SPLINE
SPL {X  -157.921, Y  +697.149, Z    +0.000, E1  +377.701, E3 -358437.505}
SPL {X  -159.579, Y  +682.959, Z    +0.000, E1  +369.793, E3 -358445.453}
SPL {X  -159.938, Y  +675.561, Z    +0.000, E1  +365.399, E3 -358447.875}
SPL {X  -159.990, Y  +669.910, Z    +0.000, E1  +361.710, E3 -358449.166}
SPL {X  -159.990, Y  +665.465, Z    +0.000, E1  +358.378, E3 -358450.084}
SPL {X  -159.990, Y  +661.791, Z    +0.000, E1  +355.213, E3 -358450.921}
SPL {X  -159.990, Y  +656.991, Z    +0.000, E1  +350.742, E3 -358452.341}
SPL {X  -159.990, Y  +648.067, Z    +0.000, E1  +342.328, E3 -358456.070}
SPL {X  -159.990, Y  +624.891, Z    +0.000, E1  +327.004, E3 -358474.558}
SPL {X  -159.990, Y  +618.109, Z    +0.000, E1  +324.631, E3 -358482.734}
SPL {X  -159.990, Y  +591.256, Z    +0.000, E1  +319.966, E3 -358526.411}
SPL {X  -159.990, Y  +586.740, Z    +0.000, E1  +319.956, E3 -358537.801}
SPL {X  -159.990, Y  +581.814, Z    +0.000, E1  +319.956, E3 -358550.241}
SPL {X  -159.990, Y  +577.274, Z    +0.000, E1  +319.964, E3 -358561.718}
SPL {X  -159.990, Y  +572.933, Z    +0.000, E1  +319.959, E3 -358572.660}
SPL {X  -159.990, Y  +568.504, Z    +0.000, E1  +319.956, E3 -358583.822}
SPL {X  -159.990, Y  +564.427, Z    +0.000, E1  +319.959, E3 -358594.108}
SPL {X  -159.990, Y  +558.823, Z    +0.000, E1  +319.916, E3 -358608.188}
SPL {X  -159.990, Y  +553.571, Z    +0.000, E1  +319.954, E3 -358621.469}
SPL {X  -159.990, Y  +549.413, Z    +0.000, E1  +319.938, E3 -358631.935}
SPL {X  -159.990, Y  +543.439, Z    +0.000, E1  +319.921, E3 -358647.023}
SPL {X  -159.990, Y  +537.213, Z    +0.000, E1  +319.937, E3 -358662.766}
SPL {X  -159.990, Y  +532.291, Z    +0.000, E1  +319.951, E3 -358675.191}
SPL {X  -159.990, Y  +527.393, Z    +0.000, E1  +319.924, E3 -358687.500}
SPL {X  -159.990, Y  +522.533, Z    +0.000, E1  +319.951, E3 -358699.797}
SPL {X  -159.990, Y  +502.378, Z    +0.000, E1  +313.079, E3 -358704.201}
SPL {X  -159.990, Y  +493.568, Z    +0.000, E1  +312.053, E3 -358715.369}
SPL {X  -159.990, Y  +489.464, Z    +0.000, E1  +313.059, E3 -358729.235}
SPL {X  -159.990, Y  +484.831, Z    +0.000, E1  +314.066, E3 -358744.769}
SPL {X  -159.990, Y  +480.580, Z    +0.000, E1  +315.242, E3 -358760.455}
SPL {X  -159.990, Y  +476.546, Z    +0.000, E1  +316.165, E3 -358774.750}
SPL {X  -159.990, Y  +472.671, Z    +0.000, E1  +317.192, E3 -358789.577}
SPL {X  -159.990, Y  +468.809, Z    +0.000, E1  +318.343, E3 -358805.506}
SPL {X  -159.990, Y  +465.057, Z    +0.000, E1  +319.375, E3 -358820.664}
SPL {X  -159.990, Y  +461.409, Z    +0.000, E1  +319.848, E3 -358832.564}
SPL {X  -159.990, Y  +456.934, Z    +0.000, E1  +319.854, E3 -358843.839}
SPL {X  -159.990, Y  +452.940, Z    +0.000, E1  +319.854, E3 -358853.884}
SPL {X  -159.990, Y  +448.856, Z    +0.000, E1  +319.859, E3 -358864.167}
SPL {X  -159.990, Y  +444.973, Z    +0.000, E1  +319.856, E3 -358873.933}
SPL {X  -159.990, Y  +439.927, Z    +0.000, E1  +319.837, E3 -358886.589}
SPL {X  -159.990, Y  +435.246, Z    +0.000, E1  +319.853, E3 -358898.398}
SPL {X  -159.990, Y  +430.690, Z    +0.000, E1  +319.854, E3 -358909.860}
SPL {X  -159.990, Y  +426.145, Z    +0.000, E1  +319.853, E3 -358921.300}
SPL {X  -159.990, Y  +421.880, Z    +0.000, E1  +319.860, E3 -358932.033}
SPL {X  -159.990, Y  +416.246, Z    +0.000, E1  +319.819, E3 -358946.162}
SPL {X  -159.990, Y  +409.936, Z    +0.000, E1  +319.849, E3 -358962.098}
SPL {X  -159.990, Y  +404.988, Z    +0.000, E1  +319.861, E3 -358974.564}
SPL {X  -159.990, Y  +400.535, Z    +0.000, E1  +319.859, E3 -358985.762}
SPL {X  -159.990, Y  +396.024, Z    +0.000, E1  +319.860, E3 -358997.118}
SPL {X  -159.990, Y  +391.614, Z    +0.000, E1  +319.860, E3 -359008.212}
SPL {X  -159.990, Y  +387.212, Z    +0.000, E1  +319.859, E3 -359019.284}
SPL {X  -159.990, Y  +382.743, Z    +0.000, E1  +319.857, E3 -359030.526}
SPL {X  -159.925, Y  +377.946, Z    +0.000, E1  +319.864, E3 -359042.662}
SPL {X  -159.703, Y  +372.915, Z    +0.000, E1  +319.904, E3 -359055.562}
SPL {X  -159.358, Y  +368.290, Z    +0.000, E1  +319.961, E3 -359067.525}
SPL {X  -158.955, Y  +364.333, Z    +0.000, E1  +320.046, E3 -359077.927}
SPL {X  -158.270, Y  +359.106, Z    +0.000, E1  +320.118, E3 -359091.738}
SPL {X  -157.143, Y  +352.453, Z    +0.000, E1  +320.322, E3 -359109.669}
SPL {X  -156.148, Y  +347.650, Z    +0.000, E1  +320.549, E3 -359122.855}
SPL {X  -155.268, Y  +343.918, Z    +0.000, E1  +320.696, E3 -359133.136}
SPL {X  -153.936, Y  +338.906, Z    +0.000, E1  +320.911, E3 -359147.075}
SPL {X  -152.628, Y  +334.526, Z    +0.000, E1  +321.188, E3 -359159.477}
SPL {X  -151.010, Y  +329.654, Z    +0.000, E1  +326.674, E3 -359217.313}
ENDSPLINE

SPLINE
SPL {X  -157.513, Y  +354.453, Z    +0.000, E1  +340.941, E3 -359263.348}
SPL {X  -159.408, Y  +368.861, Z    +0.000, E1  +348.865, E3 -359272.770}
SPL {X  -159.941, Y  +378.532, Z    +0.000, E1  +354.551, E3 -359276.376}
SPL {X  -159.990, Y  +383.966, Z    +0.000, E1  +358.149, E3 -359277.828}
SPL {X  -159.990, Y  +388.001, Z    +0.000, E1  +361.086, E3 -359278.763}
SPL {X  -159.990, Y  +392.647, Z    +0.000, E1  +364.974, E3 -359279.902}
SPL {X  -159.990, Y  +397.943, Z    +0.000, E1  +369.963, E3 -359281.486}
SPL {X  -159.990, Y  +407.689, Z    +0.000, E1  +378.860, E3 -359286.141}
SPL {X  -159.990, Y  +434.822, Z    +0.000, E1  +394.625, E3 -359310.685}
SPL {X  -159.990, Y  +460.330, Z    +0.000, E1  +398.908, E3 -359354.960}
SPL {X  -159.990, Y  +464.953, Z    +0.000, E1  +398.907, E3 -359367.118}
SPL {X  -159.990, Y  +469.353, Z    +0.000, E1  +398.902, E3 -359378.699}
SPL {X  -159.990, Y  +475.034, Z    +0.000, E1  +398.936, E3 -359393.614}
SPL {X  -159.990, Y  +481.308, Z    +0.000, E1  +398.917, E3 -359410.125}
SPL {X  -159.990, Y  +485.396, Z    +0.000, E1  +398.893, E3 -359420.884}
SPL {X  -159.990, Y  +488.362, Z    +0.000, E1  +398.896, E3 -359428.668}
SPL {X  -159.990, Y  +492.629, Z    +0.000, E1  +398.922, E3 -359439.839}
SPL {X  -159.990, Y  +497.431, Z    +0.000, E1  +398.905, E3 -359452.505}
SPL {X  -159.990, Y  +502.093, Z    +0.000, E1  +398.909, E3 -359464.780}
SPL {X  -159.990, Y  +507.821, Z    +0.000, E1  +398.930, E3 -359479.800}
SPL {X  -159.990, Y  +513.533, Z    +0.000, E1  +398.910, E3 -359494.859}
SPL {X  -159.990, Y  +519.462, Z    +0.000, E1  +398.933, E3 -359510.412}
SPL {X  -159.990, Y  +524.415, Z    +0.000, E1  +398.896, E3 -359523.476}
SPL {X  -159.990, Y  +528.627, Z    +0.000, E1  +398.910, E3 -359534.536}
SPL {X  -159.990, Y  +533.053, Z    +0.000, E1  +398.899, E3 -359546.194}
SPL {X  -159.990, Y  +537.174, Z    +0.000, E1  +398.910, E3 -359557.008}
SPL {X  -159.990, Y  +541.259, Z    +0.000, E1  +398.888, E3 -359567.808}
SPL {X  -159.990, Y  +545.676, Z    +0.000, E1  +398.913, E3 -359579.379}
SPL {X  -159.990, Y  +550.777, Z    +0.000, E1  +398.906, E3 -359592.798}
SPL {X  -159.990, Y  +554.638, Z    +0.000, E1  +398.890, E3 -359602.969}
SPL {X  -159.990, Y  +557.678, Z    +0.000, E1  +398.893, E3 -359610.945}
SPL {X  -159.990, Y  +561.696, Z    +0.000, E1  +398.912, E3 -359621.470}
SPL {X  -159.990, Y  +566.650, Z    +0.000, E1  +398.917, E3 -359634.484}
SPL {X  -159.990, Y  +571.814, Z    +0.000, E1  +398.914, E3 -359648.086}
SPL {X  -159.990, Y  +577.636, Z    +0.000, E1  +398.929, E3 -359663.384}
SPL {X  -159.990, Y  +583.167, Z    +0.000, E1  +398.906, E3 -359677.959}
SPL {X  -159.990, Y  +589.106, Z    +0.000, E1  +398.939, E3 -359693.527}
SPL {X  -159.990, Y  +594.201, Z    +0.000, E1  +398.894, E3 -359706.995}
SPL {X  -159.990, Y  +599.478, Z    +0.000, E1  +398.941, E3 -359720.799}
SPL {X  -159.990, Y  +606.904, Z    +0.000, E1  +398.953, E3 -359740.312}
SPL {X  -159.990, Y  +614.125, Z    +0.000, E1  +398.936, E3 -359759.324}
SPL {X  -159.990, Y  +619.061, Z    +0.000, E1  +398.894, E3 -359772.356}
SPL {X  -159.990, Y  +623.264, Z    +0.000, E1  +398.906, E3 -359783.405}
SPL {X  -159.990, Y  +628.669, Z    +0.000, E1  +398.928, E3 -359797.573}
SPL {X  -159.990, Y  +634.089, Z    +0.000, E1  +398.907, E3 -359811.849}
SPL {X  -159.990, Y  +638.639, Z    +0.000, E1  +398.904, E3 -359823.834}
SPL {X  -159.990, Y  +643.555, Z    +0.000, E1  +398.910, E3 -359836.754}
SPL {X  -159.990, Y  +649.380, Z    +0.000, E1  +398.930, E3 -359852.032}
SPL {X  -159.990, Y  +654.813, Z    +0.000, E1  +398.905, E3 -359866.356}
SPL {X  -159.990, Y  +658.715, Z    +0.000, E1  +398.892, E3 -359876.637}
SPL {X  -159.990, Y  +661.848, Z    +0.000, E1  +398.892, E3 -359884.876}
SPL {X  -159.990, Y  +665.703, Z    +0.000, E1  +398.903, E3 -359894.995}
SPL {X  -159.990, Y  +669.966, Z    +0.000, E1  +398.902, E3 -359906.202}
SPL {X  -159.954, Y  +674.895, Z    +0.000, E1  +398.910, E3 -359919.181}
SPL {X  -159.761, Y  +680.061, Z    +0.000, E1  +398.873, E3 -359932.960}
SPL {X  -159.443, Y  +684.716, Z    +0.000, E1  +398.815, E3 -359945.526}
SPL {X  -158.962, Y  +689.604, Z    +0.000, E1  +398.740, E3 -359958.895}
SPL {X  -158.318, Y  +694.567, Z    +0.000, E1  +398.614, E3 -359972.656}
SPL {X  -157.472, Y  +699.775, Z    +0.000, E1  +398.483, E3 -359987.216}
SPL {X  -156.506, Y  +704.705, Z    +0.000, E1  +398.294, E3 -360001.216}
SPL {X  -155.680, Y  +708.387, Z    +0.000, E1  +398.127, E3 -360011.787}
SPL {X  -154.586, Y  +712.730, Z    +0.000, E1  +397.967, E3 -360024.284}
SPL {X  -153.345, Y  +717.131, Z    +0.000, E1  +397.713, E3 -360037.168}
SPL {X  -151.080, Y  +724.146, Z    +0.000, E1  +393.201, E3 -360095.622}
ENDSPLINE

SPLINE
SPL {X  -157.921, Y  +697.149, Z    +0.000, E1  +377.701, E3 -360147.182}
SPL {X  -159.579, Y  +682.959, Z    +0.000, E1  +369.793, E3 -360155.131}
SPL {X  -159.938, Y  +675.561, Z    +0.000, E1  +365.399, E3 -360157.553}
SPL {X  -159.990, Y  +669.910, Z    +0.000, E1  +361.710, E3 -360158.844}
SPL {X  -159.990, Y  +665.465, Z    +0.000, E1  +358.378, E3 -360159.761}
SPL {X  -159.990, Y  +661.791, Z    +0.000, E1  +355.213, E3 -360160.599}
SPL {X  -159.990, Y  +656.991, Z    +0.000, E1  +350.742, E3 -360162.018}
SPL {X  -159.990, Y  +649.722, Z    +0.000, E1  +343.777, E3 -360164.937}
SPL {X  -159.990, Y  +645.752, Z    +0.000, E1  +340.157, E3 -360166.878}
SPL {X  -159.990, Y  +620.451, Z    +0.000, E1  +325.419, E3 -360189.595}
SPL {X  -159.990, Y  +591.256, Z    +0.000, E1  +319.966, E3 -360236.088}
SPL {X  -159.990, Y  +586.740, Z    +0.000, E1  +319.956, E3 -360247.479}
SPL {X  -159.990, Y  +581.814, Z    +0.000, E1  +319.956, E3 -360259.918}
SPL {X  -159.990, Y  +577.274, Z    +0.000, E1  +319.964, E3 -360271.396}
SPL {X  -159.990, Y  +572.933, Z    +0.000, E1  +319.959, E3 -360282.337}
SPL {X  -159.990, Y  +568.504, Z    +0.000, E1  +319.956, E3 -360293.500}
SPL {X  -159.990, Y  +563.189, Z    +0.000, E1  +319.932, E3 -360306.873}
SPL {X  -159.990, Y  +557.707, Z    +0.000, E1  +319.949, E3 -360320.728}
SPL {X  -159.990, Y  +552.104, Z    +0.000, E1  +319.922, E3 -360334.803}
SPL {X  -159.990, Y  +545.912, Z    +0.000, E1  +319.929, E3 -360350.453}
SPL {X  -159.990, Y  +540.054, Z    +0.000, E1  +319.939, E3 -360365.280}
SPL {X  -159.990, Y  +533.683, Z    +0.000, E1  +319.916, E3 -360381.305}
SPL {X  -159.990, Y  +527.393, Z    +0.000, E1  +319.924, E3 -360397.177}
SPL {X  -159.990, Y  +522.533, Z    +0.000, E1  +319.951, E3 -360409.475}
SPL {X  -159.990, Y  +496.806, Z    +0.000, E1  +312.216, E3 -360419.682}
SPL {X  -159.990, Y  +490.245, Z    +0.000, E1  +312.831, E3 -360436.214}
SPL {X  -159.990, Y  +486.737, Z    +0.000, E1  +313.729, E3 -360448.220}
SPL {X  -159.990, Y  +483.955, Z    +0.000, E1  +314.316, E3 -360457.512}
SPL {X  -159.990, Y  +479.762, Z    +0.000, E1  +315.381, E3 -360472.903}
SPL {X  -159.990, Y  +474.562, Z    +0.000, E1  +316.600, E3 -360491.572}
SPL {X  -159.990, Y  +470.788, Z    +0.000, E1  +317.853, E3 -360507.455}
SPL {X  -159.990, Y  +467.944, Z    +0.000, E1  +318.635, E3 -360518.776}
SPL {X  -159.990, Y  +465.057, Z    +0.000, E1  +319.375, E3 -360530.342}
SPL {X  -159.990, Y  +461.409, Z    +0.000, E1  +319.848, E3 -360542.241}
SPL {X  -159.990, Y  +456.934, Z    +0.000, E1  +319.854, E3 -360553.517}
SPL {X  -159.990, Y  +452.940, Z    +0.000, E1  +319.854, E3 -360563.562}
SPL {X  -159.990, Y  +448.856, Z    +0.000, E1  +319.859, E3 -360573.845}
SPL {X  -159.990, Y  +444.973, Z    +0.000, E1  +319.856, E3 -360583.610}
SPL {X  -159.990, Y  +439.927, Z    +0.000, E1  +319.837, E3 -360596.267}
SPL {X  -159.990, Y  +435.246, Z    +0.000, E1  +319.853, E3 -360608.076}
SPL {X  -159.990, Y  +430.690, Z    +0.000, E1  +319.854, E3 -360619.538}
SPL {X  -159.990, Y  +426.145, Z    +0.000, E1  +319.853, E3 -360630.977}
SPL {X  -159.990, Y  +421.880, Z    +0.000, E1  +319.860, E3 -360641.710}
SPL {X  -159.990, Y  +416.246, Z    +0.000, E1  +319.819, E3 -360655.839}
SPL {X  -159.990, Y  +409.936, Z    +0.000, E1  +319.849, E3 -360671.776}
SPL {X  -159.990, Y  +404.988, Z    +0.000, E1  +319.861, E3 -360684.241}
SPL {X  -159.990, Y  +400.535, Z    +0.000, E1  +319.859, E3 -360695.440}
SPL {X  -159.990, Y  +396.024, Z    +0.000, E1  +319.860, E3 -360706.796}
SPL {X  -159.990, Y  +391.614, Z    +0.000, E1  +319.860, E3 -360717.889}
SPL {X  -159.990, Y  +387.212, Z    +0.000, E1  +319.859, E3 -360728.961}
SPL {X  -159.990, Y  +382.743, Z    +0.000, E1  +319.857, E3 -360740.203}
SPL {X  -159.925, Y  +377.946, Z    +0.000, E1  +319.864, E3 -360752.340}
SPL {X  -159.703, Y  +372.915, Z    +0.000, E1  +319.904, E3 -360765.240}
SPL {X  -159.358, Y  +368.290, Z    +0.000, E1  +319.961, E3 -360777.202}
SPL {X  -158.955, Y  +364.333, Z    +0.000, E1  +320.046, E3 -360787.605}
SPL {X  -158.482, Y  +360.589, Z    +0.000, E1  +320.125, E3 -360797.531}
SPL {X  -157.729, Y  +355.695, Z    +0.000, E1  +320.237, E3 -360810.603}
SPL {X  -156.893, Y  +351.173, Z    +0.000, E1  +320.410, E3 -360822.887}
SPL {X  -156.148, Y  +347.650, Z    +0.000, E1  +320.549, E3 -360832.533}
SPL {X  -155.268, Y  +343.918, Z    +0.000, E1  +320.696, E3 -360842.814}
SPL {X  -154.153, Y  +339.677, Z    +0.000, E1  +320.896, E3 -360854.620}
SPL {X  -152.885, Y  +335.352, Z    +0.000, E1  +321.114, E3 -360866.775}
SPL {X  -151.010, Y  +329.654, Z    +0.000, E1  +326.674, E3 -360926.991}
ENDSPLINE

SPLINE
SPL {X  -157.513, Y  +354.453, Z    +0.000, E1  +340.941, E3 -360973.025}
SPL {X  -159.408, Y  +368.861, Z    +0.000, E1  +348.865, E3 -360982.448}
SPL {X  -159.941, Y  +378.532, Z    +0.000, E1  +354.551, E3 -360986.053}
SPL {X  -159.990, Y  +383.966, Z    +0.000, E1  +358.149, E3 -360987.505}
SPL {X  -159.990, Y  +389.165, Z    +0.000, E1  +361.929, E3 -360988.707}
SPL {X  -159.990, Y  +396.368, Z    +0.000, E1  +368.359, E3 -360990.679}
SPL {X  -159.990, Y  +407.689, Z    +0.000, E1  +378.860, E3 -360995.818}
SPL {X  -159.990, Y  +434.822, Z    +0.000, E1  +394.625, E3 -361020.362}
SPL {X  -159.990, Y  +460.330, Z    +0.000, E1  +398.908, E3 -361064.638}
SPL {X  -159.990, Y  +464.953, Z    +0.000, E1  +398.907, E3 -361076.796}
SPL {X  -159.990, Y  +469.353, Z    +0.000, E1  +398.902, E3 -361088.376}
SPL {X  -159.990, Y  +473.222, Z    +0.000, E1  +398.891, E3 -361098.585}
SPL {X  -159.990, Y  +477.957, Z    +0.000, E1  +398.922, E3 -361110.990}
SPL {X  -159.990, Y  +482.463, Z    +0.000, E1  +398.891, E3 -361122.877}
SPL {X  -159.990, Y  +486.996, Z    +0.000, E1  +398.928, E3 -361134.710}
SPL {X  -159.990, Y  +492.629, Z    +0.000, E1  +398.922, E3 -361149.516}
SPL {X  -159.990, Y  +497.431, Z    +0.000, E1  +398.905, E3 -361162.183}
SPL {X  -159.990, Y  +502.093, Z    +0.000, E1  +398.909, E3 -361174.457}
SPL {X  -159.990, Y  +507.821, Z    +0.000, E1  +398.930, E3 -361189.477}
SPL {X  -159.990, Y  +513.533, Z    +0.000, E1  +398.910, E3 -361204.537}
SPL {X  -159.990, Y  +518.435, Z    +0.000, E1  +398.905, E3 -361217.432}
SPL {X  -159.990, Y  +523.478, Z    +0.000, E1  +398.918, E3 -361230.660}
SPL {X  -159.990, Y  +528.627, Z    +0.000, E1  +398.910, E3 -361244.214}
SPL {X  -159.990, Y  +534.392, Z    +0.000, E1  +398.932, E3 -361259.344}
SPL {X  -159.990, Y  +540.299, Z    +0.000, E1  +398.912, E3 -361274.919}
SPL {X  -159.990, Y  +545.676, Z    +0.000, E1  +398.913, E3 -361289.056}
SPL {X  -159.990, Y  +550.777, Z    +0.000, E1  +398.906, E3 -361302.475}
SPL {X  -159.990, Y  +556.271, Z    +0.000, E1  +398.927, E3 -361316.878}
SPL {X  -159.990, Y  +561.696, Z    +0.000, E1  +398.912, E3 -361331.148}
SPL {X  -159.990, Y  +566.650, Z    +0.000, E1  +398.917, E3 -361344.161}
SPL {X  -159.990, Y  +571.814, Z    +0.000, E1  +398.914, E3 -361357.764}
SPL {X  -159.990, Y  +577.636, Z    +0.000, E1  +398.929, E3 -361373.061}
SPL {X  -159.990, Y  +583.167, Z    +0.000, E1  +398.906, E3 -361387.637}
SPL {X  -159.990, Y  +589.106, Z    +0.000, E1  +398.939, E3 -361403.204}
SPL {X  -159.990, Y  +596.185, Z    +0.000, E1  +398.945, E3 -361421.813}
SPL {X  -159.990, Y  +602.727, Z    +0.000, E1  +398.920, E3 -361439.052}
SPL {X  -159.990, Y  +608.112, Z    +0.000, E1  +398.911, E3 -361453.226}
SPL {X  -159.990, Y  +614.125, Z    +0.000, E1  +398.936, E3 -361469.002}
SPL {X  -159.990, Y  +619.061, Z    +0.000, E1  +398.894, E3 -361482.033}
SPL {X  -159.990, Y  +623.264, Z    +0.000, E1  +398.906, E3 -361493.082}
SPL {X  -159.990, Y  +628.669, Z    +0.000, E1  +398.928, E3 -361507.250}
SPL {X  -159.990, Y  +634.089, Z    +0.000, E1  +398.907, E3 -361521.526}
SPL {X  -159.990, Y  +638.639, Z    +0.000, E1  +398.904, E3 -361533.512}
SPL {X  -159.990, Y  +644.750, Z    +0.000, E1  +398.946, E3 -361549.517}
SPL {X  -159.990, Y  +650.458, Z    +0.000, E1  +398.900, E3 -361564.590}
SPL {X  -159.990, Y  +654.813, Z    +0.000, E1  +398.905, E3 -361576.034}
SPL {X  -159.990, Y  +660.353, Z    +0.000, E1  +398.930, E3 -361590.565}
SPL {X  -159.990, Y  +665.703, Z    +0.000, E1  +398.903, E3 -361604.672}
SPL {X  -159.990, Y  +671.472, Z    +0.000, E1  +398.942, E3 -361619.777}
SPL {X  -159.920, Y  +676.216, Z    +0.000, E1  +398.875, E3 -361632.412}
SPL {X  -159.761, Y  +680.061, Z    +0.000, E1  +398.873, E3 -361642.638}
SPL {X  -159.443, Y  +684.716, Z    +0.000, E1  +398.815, E3 -361655.203}
SPL {X  -158.962, Y  +689.604, Z    +0.000, E1  +398.740, E3 -361668.572}
SPL {X  -158.318, Y  +694.567, Z    +0.000, E1  +398.614, E3 -361682.333}
SPL {X  -157.472, Y  +699.775, Z    +0.000, E1  +398.483, E3 -361696.893}
SPL {X  -156.506, Y  +704.705, Z    +0.000, E1  +398.294, E3 -361710.893}
SPL {X  -155.357, Y  +709.721, Z    +0.000, E1  +398.108, E3 -361725.248}
SPL {X  -154.005, Y  +714.851, Z    +0.000, E1  +397.854, E3 -361740.143}
SPL {X  -153.100, Y  +717.944, Z    +0.000, E1  +397.652, E3 -361749.253}
SPL {X  -151.080, Y  +724.146, Z    +0.000, E1  +393.201, E3 -361805.299}
ENDSPLINE

SPLINE
SPL {X  -157.921, Y  +697.149, Z    +0.000, E1  +377.701, E3 -361856.860}
SPL {X  -159.579, Y  +682.959, Z    +0.000, E1  +369.793, E3 -361864.808}
SPL {X  -159.938, Y  +675.561, Z    +0.000, E1  +365.399, E3 -361867.230}
SPL {X  -159.990, Y  +669.910, Z    +0.000, E1  +361.710, E3 -361868.521}
SPL {X  -159.990, Y  +665.465, Z    +0.000, E1  +358.378, E3 -361869.439}
SPL {X  -159.990, Y  +661.791, Z    +0.000, E1  +355.213, E3 -361870.276}
SPL {X  -159.990, Y  +656.991, Z    +0.000, E1  +350.742, E3 -361871.696}
SPL {X  -159.990, Y  +649.722, Z    +0.000, E1  +343.777, E3 -361874.614}
SPL {X  -159.990, Y  +645.752, Z    +0.000, E1  +340.157, E3 -361876.555}
SPL {X  -159.990, Y  +620.451, Z    +0.000, E1  +325.419, E3 -361899.272}
SPL {X  -159.990, Y  +591.256, Z    +0.000, E1  +319.966, E3 -361945.766}
SPL {X  -159.990, Y  +586.740, Z    +0.000, E1  +319.956, E3 -361957.156}
SPL {X  -159.990, Y  +581.814, Z    +0.000, E1  +319.956, E3 -361969.596}
SPL {X  -159.990, Y  +577.274, Z    +0.000, E1  +319.964, E3 -361981.073}
SPL {X  -159.990, Y  +572.933, Z    +0.000, E1  +319.959, E3 -361992.014}
SPL {X  -159.990, Y  +568.504, Z    +0.000, E1  +319.956, E3 -362003.177}
SPL {X  -159.990, Y  +563.189, Z    +0.000, E1  +319.932, E3 -362016.550}
SPL {X  -159.990, Y  +557.707, Z    +0.000, E1  +319.949, E3 -362030.406}
SPL {X  -159.990, Y  +552.104, Z    +0.000, E1  +319.922, E3 -362044.481}
SPL {X  -159.990, Y  +545.912, Z    +0.000, E1  +319.929, E3 -362060.130}
SPL {X  -159.990, Y  +540.054, Z    +0.000, E1  +319.939, E3 -362074.957}
SPL {X  -159.990, Y  +533.683, Z    +0.000, E1  +319.916, E3 -362090.982}
SPL {X  -159.990, Y  +527.393, Z    +0.000, E1  +319.924, E3 -362106.855}
SPL {X  -159.990, Y  +522.533, Z    +0.000, E1  +319.951, E3 -362119.152}
SPL {X  -159.990, Y  +502.378, Z    +0.000, E1  +313.079, E3 -362123.556}
SPL {X  -159.990, Y  +493.568, Z    +0.000, E1  +312.053, E3 -362134.724}
SPL {X  -159.990, Y  +488.437, Z    +0.000, E1  +313.241, E3 -362151.939}
SPL {X  -159.990, Y  +483.955, Z    +0.000, E1  +314.316, E3 -362167.189}
SPL {X  -159.990, Y  +480.580, Z    +0.000, E1  +315.242, E3 -362179.810}
SPL {X  -159.990, Y  +476.546, Z    +0.000, E1  +316.165, E3 -362194.105}
SPL {X  -159.990, Y  +472.671, Z    +0.000, E1  +317.192, E3 -362208.932}
SPL {X  -159.990, Y  +468.809, Z    +0.000, E1  +318.343, E3 -362224.861}
SPL {X  -159.990, Y  +465.057, Z    +0.000, E1  +319.375, E3 -362240.019}
SPL {X  -159.990, Y  +461.409, Z    +0.000, E1  +319.848, E3 -362251.919}
SPL {X  -159.990, Y  +456.934, Z    +0.000, E1  +319.854, E3 -362263.194}
SPL {X  -159.990, Y  +452.940, Z    +0.000, E1  +319.854, E3 -362273.239}
SPL {X  -159.990, Y  +448.856, Z    +0.000, E1  +319.859, E3 -362283.522}
SPL {X  -159.990, Y  +443.741, Z    +0.000, E1  +319.827, E3 -362296.340}
SPL {X  -159.990, Y  +436.703, Z    +0.000, E1  +319.809, E3 -362314.022}
SPL {X  -159.990, Y  +430.690, Z    +0.000, E1  +319.854, E3 -362329.215}
SPL {X  -159.990, Y  +426.145, Z    +0.000, E1  +319.853, E3 -362340.655}
SPL {X  -159.990, Y  +421.880, Z    +0.000, E1  +319.860, E3 -362351.388}
SPL {X  -159.990, Y  +417.572, Z    +0.000, E1  +319.852, E3 -362362.215}
SPL {X  -159.990, Y  +412.619, Z    +0.000, E1  +319.850, E3 -362374.706}
SPL {X  -159.990, Y  +406.264, Z    +0.000, E1  +319.825, E3 -362390.654}
SPL {X  -159.990, Y  +400.535, Z    +0.000, E1  +319.859, E3 -362405.117}
SPL {X  -159.990, Y  +396.024, Z    +0.000, E1  +319.860, E3 -362416.473}
SPL {X  -159.990, Y  +391.614, Z    +0.000, E1  +319.860, E3 -362427.567}
SPL {X  -159.990, Y  +387.212, Z    +0.000, E1  +319.859, E3 -362438.639}
SPL {X  -159.990, Y  +382.743, Z    +0.000, E1  +319.857, E3 -362449.880}
SPL {X  -159.925, Y  +377.946, Z    +0.000, E1  +319.864, E3 -362462.017}
SPL {X  -159.703, Y  +372.915, Z    +0.000, E1  +319.904, E3 -362474.917}
SPL {X  -159.358, Y  +368.290, Z    +0.000, E1  +319.961, E3 -362486.880}
SPL {X  -158.955, Y  +364.333, Z    +0.000, E1  +320.046, E3 -362497.282}
SPL {X  -158.482, Y  +360.589, Z    +0.000, E1  +320.125, E3 -362507.208}
SPL {X  -157.729, Y  +355.695, Z    +0.000, E1  +320.237, E3 -362520.281}
SPL {X  -156.893, Y  +351.173, Z    +0.000, E1  +320.410, E3 -362532.564}
SPL {X  -156.148, Y  +347.650, Z    +0.000, E1  +320.549, E3 -362542.210}
SPL {X  -155.268, Y  +343.918, Z    +0.000, E1  +320.696, E3 -362552.491}
SPL {X  -154.153, Y  +339.677, Z    +0.000, E1  +320.896, E3 -362564.298}
SPL {X  -152.885, Y  +335.352, Z    +0.000, E1  +321.114, E3 -362576.452}
SPL {X  -151.010, Y  +329.654, Z    +0.000, E1  +326.674, E3 -362636.668}
ENDSPLINE

SPLINE
SPL {X  -157.513, Y  +354.453, Z    +0.000, E1  +340.941, E3 -362682.703}
SPL {X  -159.638, Y  +371.886, Z    +0.000, E1  +350.545, E3 -362693.365}
SPL {X  -159.990, Y  +382.357, Z    +0.000, E1  +356.972, E3 -362696.780}
SPL {X  -159.990, Y  +389.165, Z    +0.000, E1  +361.929, E3 -362698.385}
SPL {X  -159.990, Y  +396.368, Z    +0.000, E1  +368.359, E3 -362700.357}
SPL {X  -159.990, Y  +407.689, Z    +0.000, E1  +378.860, E3 -362705.496}
SPL {X  -159.990, Y  +434.822, Z    +0.000, E1  +394.625, E3 -362730.040}
SPL {X  -159.990, Y  +460.330, Z    +0.000, E1  +398.908, E3 -362774.315}
SPL {X  -159.990, Y  +464.953, Z    +0.000, E1  +398.907, E3 -362786.473}
SPL {X  -159.990, Y  +469.353, Z    +0.000, E1  +398.902, E3 -362798.054}
SPL {X  -159.990, Y  +475.034, Z    +0.000, E1  +398.936, E3 -362812.969}
SPL {X  -159.990, Y  +481.308, Z    +0.000, E1  +398.917, E3 -362829.479}
SPL {X  -159.990, Y  +485.396, Z    +0.000, E1  +398.893, E3 -362840.239}
SPL {X  -159.990, Y  +488.362, Z    +0.000, E1  +398.896, E3 -362848.022}
SPL {X  -159.990, Y  +492.629, Z    +0.000, E1  +398.922, E3 -362859.194}
SPL {X  -159.990, Y  +497.431, Z    +0.000, E1  +398.905, E3 -362871.860}
SPL {X  -159.990, Y  +502.093, Z    +0.000, E1  +398.909, E3 -362884.135}
SPL {X  -159.990, Y  +507.821, Z    +0.000, E1  +398.930, E3 -362899.155}
SPL {X  -159.990, Y  +513.533, Z    +0.000, E1  +398.910, E3 -362914.214}
SPL {X  -159.990, Y  +518.435, Z    +0.000, E1  +398.905, E3 -362927.109}
SPL {X  -159.990, Y  +523.478, Z    +0.000, E1  +398.918, E3 -362940.338}
SPL {X  -159.990, Y  +528.627, Z    +0.000, E1  +398.910, E3 -362953.891}
SPL {X  -159.990, Y  +533.053, Z    +0.000, E1  +398.899, E3 -362965.549}
SPL {X  -159.990, Y  +537.174, Z    +0.000, E1  +398.910, E3 -362976.363}
SPL {X  -159.990, Y  +541.259, Z    +0.000, E1  +398.888, E3 -362987.163}
SPL {X  -159.990, Y  +545.676, Z    +0.000, E1  +398.913, E3 -362998.734}
SPL {X  -159.990, Y  +550.777, Z    +0.000, E1  +398.906, E3 -363012.153}
SPL {X  -159.990, Y  +554.638, Z    +0.000, E1  +398.890, E3 -363022.324}
SPL {X  -159.990, Y  +557.678, Z    +0.000, E1  +398.893, E3 -363030.300}
SPL {X  -159.990, Y  +561.696, Z    +0.000, E1  +398.912, E3 -363040.825}
SPL {X  -159.990, Y  +566.650, Z    +0.000, E1  +398.917, E3 -363053.839}
SPL {X  -159.990, Y  +571.814, Z    +0.000, E1  +398.914, E3 -363067.441}
SPL {X  -159.990, Y  +577.636, Z    +0.000, E1  +398.929, E3 -363082.739}
SPL {X  -159.990, Y  +583.167, Z    +0.000, E1  +398.906, E3 -363097.314}
SPL {X  -159.990, Y  +587.761, Z    +0.000, E1  +398.902, E3 -363109.399}
SPL {X  -159.990, Y  +592.962, Z    +0.000, E1  +398.925, E3 -363123.043}
SPL {X  -159.990, Y  +597.767, Z    +0.000, E1  +398.897, E3 -363135.719}
SPL {X  -159.990, Y  +602.727, Z    +0.000, E1  +398.920, E3 -363148.729}
SPL {X  -159.990, Y  +608.112, Z    +0.000, E1  +398.911, E3 -363162.904}
SPL {X  -159.990, Y  +614.125, Z    +0.000, E1  +398.936, E3 -363178.679}
SPL {X  -159.990, Y  +619.061, Z    +0.000, E1  +398.894, E3 -363191.711}
SPL {X  -159.990, Y  +623.264, Z    +0.000, E1  +398.906, E3 -363202.760}
SPL {X  -159.990, Y  +628.669, Z    +0.000, E1  +398.928, E3 -363216.928}
SPL {X  -159.990, Y  +634.089, Z    +0.000, E1  +398.907, E3 -363231.204}
SPL {X  -159.990, Y  +638.639, Z    +0.000, E1  +398.904, E3 -363243.189}
SPL {X  -159.990, Y  +643.555, Z    +0.000, E1  +398.910, E3 -363256.109}
SPL {X  -159.990, Y  +649.380, Z    +0.000, E1  +398.930, E3 -363271.387}
SPL {X  -159.990, Y  +654.813, Z    +0.000, E1  +398.905, E3 -363285.711}
SPL {X  -159.990, Y  +660.353, Z    +0.000, E1  +398.930, E3 -363300.242}
SPL {X  -159.990, Y  +665.703, Z    +0.000, E1  +398.903, E3 -363314.350}
SPL {X  -159.990, Y  +671.472, Z    +0.000, E1  +398.942, E3 -363329.454}
SPL {X  -159.920, Y  +676.216, Z    +0.000, E1  +398.875, E3 -363342.090}
SPL {X  -159.761, Y  +680.061, Z    +0.000, E1  +398.873, E3 -363352.315}
SPL {X  -159.443, Y  +684.716, Z    +0.000, E1  +398.815, E3 -363364.880}
SPL {X  -158.962, Y  +689.604, Z    +0.000, E1  +398.740, E3 -363378.250}
SPL {X  -158.318, Y  +694.567, Z    +0.000, E1  +398.614, E3 -363392.011}
SPL {X  -157.472, Y  +699.775, Z    +0.000, E1  +398.483, E3 -363406.570}
SPL {X  -156.506, Y  +704.705, Z    +0.000, E1  +398.294, E3 -363420.571}
SPL {X  -155.357, Y  +709.721, Z    +0.000, E1  +398.108, E3 -363434.926}
SPL {X  -154.286, Y  +713.838, Z    +0.000, E1  +397.877, E3 -363446.908}
SPL {X  -153.345, Y  +717.131, Z    +0.000, E1  +397.713, E3 -363456.523}
SPL {X  -151.080, Y  +724.146, Z    +0.000, E1  +393.201, E3 -363514.976}
ENDSPLINE

SPLINE
SPL {X  -157.921, Y  +697.149, Z    +0.000, E1  +377.701, E3 -363566.537}
SPL {X  -159.579, Y  +682.959, Z    +0.000, E1  +369.793, E3 -363574.486}
SPL {X  -159.938, Y  +675.561, Z    +0.000, E1  +365.399, E3 -363576.908}
SPL {X  -159.990, Y  +669.910, Z    +0.000, E1  +361.710, E3 -363578.199}
SPL {X  -159.990, Y  +665.465, Z    +0.000, E1  +358.378, E3 -363579.116}
SPL {X  -159.990, Y  +661.791, Z    +0.000, E1  +355.213, E3 -363579.954}
SPL {X  -159.990, Y  +656.991, Z    +0.000, E1  +350.742, E3 -363581.373}
SPL {X  -159.990, Y  +649.722, Z    +0.000, E1  +343.777, E3 -363584.292}
SPL {X  -159.990, Y  +645.752, Z    +0.000, E1  +340.157, E3 -363586.233}
SPL {X  -159.990, Y  +624.891, Z    +0.000, E1  +327.004, E3 -363603.591}
SPL {X  -159.990, Y  +618.109, Z    +0.000, E1  +324.631, E3 -363611.767}
SPL {X  -159.990, Y  +591.256, Z    +0.000, E1  +319.966, E3 -363655.443}
SPL {X  -159.990, Y  +586.740, Z    +0.000, E1  +319.956, E3 -363666.834}
SPL {X  -159.990, Y  +581.814, Z    +0.000, E1  +319.956, E3 -363679.273}
SPL {X  -159.990, Y  +577.274, Z    +0.000, E1  +319.964, E3 -363690.751}
SPL {X  -159.990, Y  +572.933, Z    +0.000, E1  +319.959, E3 -363701.692}
SPL {X  -159.990, Y  +568.504, Z    +0.000, E1  +319.956, E3 -363712.854}
SPL {X  -159.990, Y  +564.427, Z    +0.000, E1  +319.959, E3 -363723.140}
SPL {X  -159.990, Y  +558.823, Z    +0.000, E1  +319.916, E3 -363737.220}
SPL {X  -159.990, Y  +553.571, Z    +0.000, E1  +319.954, E3 -363750.502}
SPL {X  -159.990, Y  +549.413, Z    +0.000, E1  +319.938, E3 -363760.968}
SPL {X  -159.990, Y  +544.924, Z    +0.000, E1  +319.955, E3 -363772.349}
SPL {X  -159.990, Y  +540.054, Z    +0.000, E1  +319.939, E3 -363784.635}
SPL {X  -159.990, Y  +533.683, Z    +0.000, E1  +319.916, E3 -363800.660}
SPL {X  -159.990, Y  +528.899, Z    +0.000, E1  +319.955, E3 -363812.776}
SPL {X  -159.990, Y  +523.984, Z    +0.000, E1  +319.922, E3 -363825.122}
SPL {X  -159.990, Y  +495.402, Z    +0.000, E1  +312.238, E3 -363842.053}
SPL {X  -159.990, Y  +489.464, Z    +0.000, E1  +313.059, E3 -363858.268}
SPL {X  -159.990, Y  +484.831, Z    +0.000, E1  +314.066, E3 -363873.801}
SPL {X  -159.990, Y  +479.762, Z    +0.000, E1  +315.381, E3 -363892.258}
SPL {X  -159.990, Y  +475.871, Z    +0.000, E1  +316.362, E3 -363906.306}
SPL {X  -159.990, Y  +472.671, Z    +0.000, E1  +317.192, E3 -363918.610}
SPL {X  -159.990, Y  +468.809, Z    +0.000, E1  +318.343, E3 -363934.538}
SPL {X  -159.990, Y  +465.057, Z    +0.000, E1  +319.375, E3 -363949.697}
SPL {X  -159.990, Y  +461.409, Z    +0.000, E1  +319.848, E3 -363961.596}
SPL {X  -159.990, Y  +456.934, Z    +0.000, E1  +319.854, E3 -363972.872}
SPL {X  -159.990, Y  +452.940, Z    +0.000, E1  +319.854, E3 -363982.916}
SPL {X  -159.990, Y  +448.856, Z    +0.000, E1  +319.859, E3 -363993.200}
SPL {X  -159.990, Y  +444.973, Z    +0.000, E1  +319.856, E3 -364002.965}
SPL {X  -159.990, Y  +439.927, Z    +0.000, E1  +319.837, E3 -364015.621}
SPL {X  -159.990, Y  +435.246, Z    +0.000, E1  +319.853, E3 -364027.431}
SPL {X  -159.990, Y  +430.690, Z    +0.000, E1  +319.854, E3 -364038.893}
SPL {X  -159.990, Y  +426.145, Z    +0.000, E1  +319.853, E3 -364050.332}
SPL {X  -159.990, Y  +421.880, Z    +0.000, E1  +319.860, E3 -364061.065}
SPL {X  -159.990, Y  +417.572, Z    +0.000, E1  +319.852, E3 -364071.892}
SPL {X  -159.990, Y  +412.619, Z    +0.000, E1  +319.850, E3 -364084.383}
SPL {X  -159.990, Y  +406.264, Z    +0.000, E1  +319.825, E3 -364100.332}
SPL {X  -159.990, Y  +400.535, Z    +0.000, E1  +319.859, E3 -364114.794}
SPL {X  -159.990, Y  +396.024, Z    +0.000, E1  +319.860, E3 -364126.150}
SPL {X  -159.990, Y  +391.614, Z    +0.000, E1  +319.860, E3 -364137.244}
SPL {X  -159.990, Y  +387.212, Z    +0.000, E1  +319.859, E3 -364148.316}
SPL {X  -159.990, Y  +382.743, Z    +0.000, E1  +319.857, E3 -364159.558}
SPL {X  -159.925, Y  +377.946, Z    +0.000, E1  +319.864, E3 -364171.695}
SPL {X  -159.703, Y  +372.915, Z    +0.000, E1  +319.904, E3 -364184.594}
SPL {X  -159.358, Y  +368.290, Z    +0.000, E1  +319.961, E3 -364196.557}
SPL {X  -158.955, Y  +364.333, Z    +0.000, E1  +320.046, E3 -364206.960}
SPL {X  -158.482, Y  +360.589, Z    +0.000, E1  +320.125, E3 -364216.886}
SPL {X  -157.729, Y  +355.695, Z    +0.000, E1  +320.237, E3 -364229.958}
SPL {X  -156.893, Y  +351.173, Z    +0.000, E1  +320.410, E3 -364242.242}
SPL {X  -156.148, Y  +347.650, Z    +0.000, E1  +320.549, E3 -364251.888}
SPL {X  -155.268, Y  +343.918, Z    +0.000, E1  +320.696, E3 -364262.168}
SPL {X  -153.936, Y  +338.906, Z    +0.000, E1  +320.911, E3 -364276.108}
SPL {X  -152.628, Y  +334.526, Z    +0.000, E1  +321.188, E3 -364288.510}
SPL {X  -151.010, Y  +329.654, Z    +0.000, E1  +326.674, E3 -364346.346}
ENDSPLINE

SPLINE
SPL {X  -157.513, Y  +354.453, Z    +0.000, E1  +340.941, E3 -364392.380}
SPL {X  -159.408, Y  +368.861, Z    +0.000, E1  +348.865, E3 -364401.803}
SPL {X  -159.941, Y  +378.532, Z    +0.000, E1  +354.551, E3 -364405.408}
SPL {X  -159.990, Y  +383.966, Z    +0.000, E1  +358.149, E3 -364406.860}
SPL {X  -159.990, Y  +388.001, Z    +0.000, E1  +361.086, E3 -364407.795}
SPL {X  -159.990, Y  +392.647, Z    +0.000, E1  +364.974, E3 -364408.934}
SPL {X  -159.990, Y  +397.943, Z    +0.000, E1  +369.963, E3 -364410.519}
SPL {X  -159.990, Y  +406.530, Z    +0.000, E1  +377.917, E3 -364414.416}
SPL {X  -159.990, Y  +429.014, Z    +0.000, E1  +392.438, E3 -364433.073}
SPL {X  -159.990, Y  +437.635, Z    +0.000, E1  +395.495, E3 -364443.305}
SPL {X  -159.990, Y  +460.330, Z    +0.000, E1  +398.908, E3 -364483.992}
SPL {X  -159.990, Y  +464.953, Z    +0.000, E1  +398.907, E3 -364496.151}
SPL {X  -159.990, Y  +469.353, Z    +0.000, E1  +398.902, E3 -364507.731}
SPL {X  -159.990, Y  +475.034, Z    +0.000, E1  +398.936, E3 -364522.646}
SPL {X  -159.990, Y  +481.308, Z    +0.000, E1  +398.917, E3 -364539.157}
SPL {X  -159.990, Y  +486.996, Z    +0.000, E1  +398.928, E3 -364554.065}
SPL {X  -159.990, Y  +492.629, Z    +0.000, E1  +398.922, E3 -364568.871}
SPL {X  -159.990, Y  +497.431, Z    +0.000, E1  +398.905, E3 -364581.537}
SPL {X  -159.990, Y  +502.093, Z    +0.000, E1  +398.909, E3 -364593.812}
SPL {X  -159.990, Y  +507.821, Z    +0.000, E1  +398.930, E3 -364608.832}
SPL {X  -159.990, Y  +513.533, Z    +0.000, E1  +398.910, E3 -364623.892}
SPL {X  -159.990, Y  +518.435, Z    +0.000, E1  +398.905, E3 -364636.787}
SPL {X  -159.990, Y  +523.478, Z    +0.000, E1  +398.918, E3 -364650.015}
SPL {X  -159.990, Y  +528.627, Z    +0.000, E1  +398.910, E3 -364663.569}
SPL {X  -159.990, Y  +534.392, Z    +0.000, E1  +398.932, E3 -364678.699}
SPL {X  -159.990, Y  +540.299, Z    +0.000, E1  +398.912, E3 -364694.274}
SPL {X  -159.990, Y  +545.676, Z    +0.000, E1  +398.913, E3 -364708.411}
SPL {X  -159.990, Y  +550.777, Z    +0.000, E1  +398.906, E3 -364721.830}
SPL {X  -159.990, Y  +556.271, Z    +0.000, E1  +398.927, E3 -364736.233}
SPL {X  -159.990, Y  +561.696, Z    +0.000, E1  +398.912, E3 -364750.502}
SPL {X  -159.990, Y  +566.650, Z    +0.000, E1  +398.917, E3 -364763.516}
SPL {X  -159.990, Y  +571.814, Z    +0.000, E1  +398.914, E3 -364777.119}
SPL {X  -159.990, Y  +577.636, Z    +0.000, E1  +398.929, E3 -364792.416}
SPL {X  -159.990, Y  +583.167, Z    +0.000, E1  +398.906, E3 -364806.992}
SPL {X  -159.990, Y  +587.761, Z    +0.000, E1  +398.902, E3 -364819.077}
SPL {X  -159.990, Y  +592.962, Z    +0.000, E1  +398.925, E3 -364832.721}
SPL {X  -159.990, Y  +597.767, Z    +0.000, E1  +398.897, E3 -364845.396}
SPL {X  -159.990, Y  +602.727, Z    +0.000, E1  +398.920, E3 -364858.407}
SPL {X  -159.990, Y  +608.112, Z    +0.000, E1  +398.911, E3 -364872.581}
SPL {X  -159.990, Y  +613.039, Z    +0.000, E1  +398.906, E3 -364885.544}
SPL {X  -159.990, Y  +618.087, Z    +0.000, E1  +398.915, E3 -364898.803}
SPL {X  -159.990, Y  +623.264, Z    +0.000, E1  +398.906, E3 -364912.437}
SPL {X  -159.990, Y  +628.669, Z    +0.000, E1  +398.928, E3 -364926.605}
SPL {X  -159.990, Y  +634.089, Z    +0.000, E1  +398.907, E3 -364940.881}
SPL {X  -159.990, Y  +638.639, Z    +0.000, E1  +398.904, E3 -364952.867}
SPL {X  -159.990, Y  +643.555, Z    +0.000, E1  +398.910, E3 -364965.786}
SPL {X  -159.990, Y  +649.380, Z    +0.000, E1  +398.930, E3 -364981.064}
SPL {X  -159.990, Y  +654.813, Z    +0.000, E1  +398.905, E3 -364995.389}
SPL {X  -159.990, Y  +660.353, Z    +0.000, E1  +398.930, E3 -365009.920}
SPL {X  -159.990, Y  +665.703, Z    +0.000, E1  +398.903, E3 -365024.027}
SPL {X  -159.990, Y  +669.966, Z    +0.000, E1  +398.902, E3 -365035.234}
SPL {X  -159.954, Y  +674.895, Z    +0.000, E1  +398.910, E3 -365048.214}
SPL {X  -159.761, Y  +680.061, Z    +0.000, E1  +398.873, E3 -365061.993}
SPL {X  -159.443, Y  +684.716, Z    +0.000, E1  +398.815, E3 -365074.558}
SPL {X  -158.962, Y  +689.604, Z    +0.000, E1  +398.740, E3 -365087.927}
SPL {X  -158.318, Y  +694.567, Z    +0.000, E1  +398.614, E3 -365101.688}
SPL {X  -157.472, Y  +699.775, Z    +0.000, E1  +398.483, E3 -365116.248}
SPL {X  -156.506, Y  +704.705, Z    +0.000, E1  +398.294, E3 -365130.248}
SPL {X  -155.357, Y  +709.721, Z    +0.000, E1  +398.108, E3 -365144.603}
SPL {X  -154.005, Y  +714.851, Z    +0.000, E1  +397.854, E3 -365159.498}
SPL {X  -153.100, Y  +717.944, Z    +0.000, E1  +397.652, E3 -365168.608}
SPL {X  -151.080, Y  +724.146, Z    +0.000, E1  +393.201, E3 -365224.654}
ENDSPLINE

SPLINE
SPL {X  -157.921, Y  +697.149, Z    +0.000, E1  +377.701, E3 -365276.215}
SPL {X  -159.579, Y  +682.959, Z    +0.000, E1  +369.793, E3 -365284.163}
SPL {X  -159.938, Y  +675.561, Z    +0.000, E1  +365.399, E3 -365286.585}
SPL {X  -159.990, Y  +669.910, Z    +0.000, E1  +361.710, E3 -365287.876}
SPL {X  -159.990, Y  +665.465, Z    +0.000, E1  +358.378, E3 -365288.793}
SPL {X  -159.990, Y  +661.791, Z    +0.000, E1  +355.213, E3 -365289.631}
SPL {X  -159.990, Y  +656.991, Z    +0.000, E1  +350.742, E3 -365291.050}
SPL {X  -159.990, Y  +648.067, Z    +0.000, E1  +342.328, E3 -365294.780}
SPL {X  -159.990, Y  +620.451, Z    +0.000, E1  +325.419, E3 -365318.627}
SPL {X  -159.990, Y  +591.256, Z    +0.000, E1  +319.966, E3 -365365.121}
SPL {X  -159.990, Y  +586.740, Z    +0.000, E1  +319.956, E3 -365376.511}
SPL {X  -159.990, Y  +581.814, Z    +0.000, E1  +319.956, E3 -365388.951}
SPL {X  -159.990, Y  +577.274, Z    +0.000, E1  +319.964, E3 -365400.428}
SPL {X  -159.990, Y  +572.933, Z    +0.000, E1  +319.959, E3 -365411.369}
SPL {X  -159.990, Y  +568.504, Z    +0.000, E1  +319.956, E3 -365422.532}
SPL {X  -159.990, Y  +564.427, Z    +0.000, E1  +319.959, E3 -365432.818}
SPL {X  -159.990, Y  +558.823, Z    +0.000, E1  +319.916, E3 -365446.897}
SPL {X  -159.990, Y  +553.571, Z    +0.000, E1  +319.954, E3 -365460.179}
SPL {X  -159.990, Y  +549.413, Z    +0.000, E1  +319.938, E3 -365470.645}
SPL {X  -159.990, Y  +543.439, Z    +0.000, E1  +319.921, E3 -365485.733}
SPL {X  -159.990, Y  +537.213, Z    +0.000, E1  +319.937, E3 -365501.476}
SPL {X  -159.990, Y  +532.291, Z    +0.000, E1  +319.951, E3 -365513.901}
SPL {X  -159.990, Y  +528.899, Z    +0.000, E1  +319.955, E3 -365522.453}
SPL {X  -159.990, Y  +523.984, Z    +0.000, E1  +319.922, E3 -365534.800}
SPL {X  -159.990, Y  +496.806, Z    +0.000, E1  +312.216, E3 -365548.715}
SPL {X  -159.990, Y  +490.245, Z    +0.000, E1  +312.831, E3 -365565.246}
SPL {X  -159.990, Y  +484.831, Z    +0.000, E1  +314.066, E3 -365583.479}
SPL {X  -159.990, Y  +480.580, Z    +0.000, E1  +315.242, E3 -365599.165}
SPL {X  -159.990, Y  +476.546, Z    +0.000, E1  +316.165, E3 -365613.460}
SPL {X  -159.990, Y  +472.671, Z    +0.000, E1  +317.192, E3 -365628.287}
SPL {X  -159.990, Y  +468.809, Z    +0.000, E1  +318.343, E3 -365644.216}
SPL {X  -159.990, Y  +465.057, Z    +0.000, E1  +319.375, E3 -365659.374}
SPL {X  -159.990, Y  +461.409, Z    +0.000, E1  +319.848, E3 -365671.273}
SPL {X  -159.990, Y  +456.934, Z    +0.000, E1  +319.854, E3 -365682.549}
SPL {X  -159.990, Y  +452.940, Z    +0.000, E1  +319.854, E3 -365692.594}
SPL {X  -159.990, Y  +448.856, Z    +0.000, E1  +319.859, E3 -365702.877}
SPL {X  -159.990, Y  +443.741, Z    +0.000, E1  +319.827, E3 -365715.695}
SPL {X  -159.990, Y  +436.703, Z    +0.000, E1  +319.809, E3 -365733.377}
SPL {X  -159.990, Y  +430.690, Z    +0.000, E1  +319.854, E3 -365748.570}
SPL {X  -159.990, Y  +426.145, Z    +0.000, E1  +319.853, E3 -365760.010}
SPL {X  -159.990, Y  +421.880, Z    +0.000, E1  +319.860, E3 -365770.743}
SPL {X  -159.990, Y  +417.572, Z    +0.000, E1  +319.852, E3 -365781.569}
SPL {X  -159.990, Y  +412.619, Z    +0.000, E1  +319.850, E3 -365794.061}
SPL {X  -159.990, Y  +406.264, Z    +0.000, E1  +319.825, E3 -365810.009}
SPL {X  -159.990, Y  +400.535, Z    +0.000, E1  +319.859, E3 -365824.472}
SPL {X  -159.990, Y  +396.024, Z    +0.000, E1  +319.860, E3 -365835.828}
SPL {X  -159.990, Y  +391.614, Z    +0.000, E1  +319.860, E3 -365846.921}
SPL {X  -159.990, Y  +387.212, Z    +0.000, E1  +319.859, E3 -365857.994}
SPL {X  -159.990, Y  +382.743, Z    +0.000, E1  +319.857, E3 -365869.235}
SPL {X  -159.925, Y  +377.946, Z    +0.000, E1  +319.864, E3 -365881.372}
SPL {X  -159.703, Y  +372.915, Z    +0.000, E1  +319.904, E3 -365894.272}
SPL {X  -159.358, Y  +368.290, Z    +0.000, E1  +319.961, E3 -365906.234}
SPL {X  -158.955, Y  +364.333, Z    +0.000, E1  +320.046, E3 -365916.637}
SPL {X  -158.482, Y  +360.589, Z    +0.000, E1  +320.125, E3 -365926.563}
SPL {X  -157.729, Y  +355.695, Z    +0.000, E1  +320.237, E3 -365939.636}
SPL {X  -156.893, Y  +351.173, Z    +0.000, E1  +320.410, E3 -365951.919}
SPL {X  -156.148, Y  +347.650, Z    +0.000, E1  +320.549, E3 -365961.565}
SPL {X  -155.268, Y  +343.918, Z    +0.000, E1  +320.696, E3 -365971.846}
SPL {X  -154.153, Y  +339.677, Z    +0.000, E1  +320.896, E3 -365983.653}
SPL {X  -152.885, Y  +335.352, Z    +0.000, E1  +321.114, E3 -365995.807}
SPL {X  -151.010, Y  +329.654, Z    +0.000, E1  +326.674, E3 -366056.023}
ENDSPLINE

SPLINE
SPL {X  -157.513, Y  +354.453, Z    +0.000, E1  +340.941, E3 -366102.057}
SPL {X  -159.408, Y  +368.861, Z    +0.000, E1  +348.865, E3 -366111.480}
SPL {X  -159.941, Y  +378.532, Z    +0.000, E1  +354.551, E3 -366115.086}
SPL {X  -159.990, Y  +383.966, Z    +0.000, E1  +358.149, E3 -366116.538}
SPL {X  -159.990, Y  +388.001, Z    +0.000, E1  +361.086, E3 -366117.473}
SPL {X  -159.990, Y  +392.647, Z    +0.000, E1  +364.974, E3 -366118.611}
SPL {X  -159.990, Y  +397.943, Z    +0.000, E1  +369.963, E3 -366120.196}
SPL {X  -159.990, Y  +407.689, Z    +0.000, E1  +378.860, E3 -366124.850}
SPL {X  -159.990, Y  +434.822, Z    +0.000, E1  +394.625, E3 -366149.394}
SPL {X  -159.990, Y  +460.330, Z    +0.000, E1  +398.908, E3 -366193.670}
SPL {X  -159.990, Y  +464.953, Z    +0.000, E1  +398.907, E3 -366205.828}
SPL {X  -159.990, Y  +469.353, Z    +0.000, E1  +398.902, E3 -366217.408}
SPL {X  -159.990, Y  +473.222, Z    +0.000, E1  +398.891, E3 -366227.617}
SPL {X  -159.990, Y  +477.957, Z    +0.000, E1  +398.922, E3 -366240.022}
SPL {X  -159.990, Y  +482.463, Z    +0.000, E1  +398.891, E3 -366251.910}
SPL {X  -159.990, Y  +486.996, Z    +0.000, E1  +398.928, E3 -366263.742}
SPL {X  -159.990, Y  +492.629, Z    +0.000, E1  +398.922, E3 -366278.549}
SPL {X  -159.990, Y  +497.431, Z    +0.000, E1  +398.905, E3 -366291.215}
SPL {X  -159.990, Y  +502.093, Z    +0.000, E1  +398.909, E3 -366303.489}
SPL {X  -159.990, Y  +507.821, Z    +0.000, E1  +398.930, E3 -366318.510}
SPL {X  -159.990, Y  +513.533, Z    +0.000, E1  +398.910, E3 -366333.569}
SPL {X  -159.990, Y  +519.462, Z    +0.000, E1  +398.933, E3 -366349.122}
SPL {X  -159.990, Y  +524.415, Z    +0.000, E1  +398.896, E3 -366362.186}
SPL {X  -159.990, Y  +528.627, Z    +0.000, E1  +398.910, E3 -366373.246}
SPL {X  -159.990, Y  +534.392, Z    +0.000, E1  +398.932, E3 -366388.376}
SPL {X  -159.990, Y  +540.299, Z    +0.000, E1  +398.912, E3 -366403.951}
SPL {X  -159.990, Y  +545.676, Z    +0.000, E1  +398.913, E3 -366418.089}
SPL {X  -159.990, Y  +550.777, Z    +0.000, E1  +398.906, E3 -366431.508}
SPL {X  -159.990, Y  +556.271, Z    +0.000, E1  +398.927, E3 -366445.910}
SPL {X  -159.990, Y  +561.696, Z    +0.000, E1  +398.912, E3 -366460.180}
SPL {X  -159.990, Y  +566.650, Z    +0.000, E1  +398.917, E3 -366473.193}
SPL {X  -159.990, Y  +571.814, Z    +0.000, E1  +398.914, E3 -366486.796}
SPL {X  -159.990, Y  +577.636, Z    +0.000, E1  +398.929, E3 -366502.094}
SPL {X  -159.990, Y  +583.167, Z    +0.000, E1  +398.906, E3 -366516.669}
SPL {X  -159.990, Y  +587.761, Z    +0.000, E1  +398.902, E3 -366528.754}
SPL {X  -159.990, Y  +592.962, Z    +0.000, E1  +398.925, E3 -366542.398}
SPL {X  -159.990, Y  +597.767, Z    +0.000, E1  +398.897, E3 -366555.073}
SPL {X  -159.990, Y  +602.727, Z    +0.000, E1  +398.920, E3 -366568.084}
SPL {X  -159.990, Y  +608.112, Z    +0.000, E1  +398.911, E3 -366582.259}
SPL {X  -159.990, Y  +613.039, Z    +0.000, E1  +398.906, E3 -366595.221}
SPL {X  -159.990, Y  +618.087, Z    +0.000, E1  +398.915, E3 -366608.480}
SPL {X  -159.990, Y  +623.264, Z    +0.000, E1  +398.906, E3 -366622.114}
SPL {X  -159.990, Y  +628.669, Z    +0.000, E1  +398.928, E3 -366636.283}
SPL {X  -159.990, Y  +634.089, Z    +0.000, E1  +398.907, E3 -366650.558}
SPL {X  -159.990, Y  +638.639, Z    +0.000, E1  +398.904, E3 -366662.544}
SPL {X  -159.990, Y  +643.555, Z    +0.000, E1  +398.910, E3 -366675.464}
SPL {X  -159.990, Y  +649.380, Z    +0.000, E1  +398.930, E3 -366690.741}
SPL {X  -159.990, Y  +654.813, Z    +0.000, E1  +398.905, E3 -366705.066}
SPL {X  -159.990, Y  +660.353, Z    +0.000, E1  +398.930, E3 -366719.597}
SPL {X  -159.990, Y  +665.703, Z    +0.000, E1  +398.903, E3 -366733.705}
SPL {X  -159.990, Y  +669.966, Z    +0.000, E1  +398.902, E3 -366744.911}
SPL {X  -159.954, Y  +674.895, Z    +0.000, E1  +398.910, E3 -366757.891}
SPL {X  -159.761, Y  +680.061, Z    +0.000, E1  +398.873, E3 -366771.670}
SPL {X  -159.443, Y  +684.716, Z    +0.000, E1  +398.815, E3 -366784.235}
SPL {X  -158.962, Y  +689.604, Z    +0.000, E1  +398.740, E3 -366797.605}
SPL {X  -158.318, Y  +694.567, Z    +0.000, E1  +398.614, E3 -366811.366}
SPL {X  -157.472, Y  +699.775, Z    +0.000, E1  +398.483, E3 -366825.925}
SPL {X  -156.506, Y  +704.705, Z    +0.000, E1  +398.294, E3 -366839.926}
SPL {X  -155.680, Y  +708.387, Z    +0.000, E1  +398.127, E3 -366850.496}
SPL {X  -154.586, Y  +712.730, Z    +0.000, E1  +397.967, E3 -366862.993}
SPL {X  -153.345, Y  +717.131, Z    +0.000, E1  +397.713, E3 -366875.877}
SPL {X  -151.080, Y  +724.146, Z    +0.000, E1  +393.201, E3 -366934.331}
ENDSPLINE

SPLINE
SPL {X  -157.921, Y  +697.149, Z    +0.000, E1  +377.701, E3 -366985.892}
SPL {X  -159.579, Y  +682.959, Z    +0.000, E1  +369.793, E3 -366993.840}
SPL {X  -159.938, Y  +675.561, Z    +0.000, E1  +365.399, E3 -366996.263}
SPL {X  -159.990, Y  +669.910, Z    +0.000, E1  +361.710, E3 -366997.553}
SPL {X  -159.990, Y  +665.465, Z    +0.000, E1  +358.378, E3 -366998.471}
SPL {X  -159.990, Y  +661.791, Z    +0.000, E1  +355.213, E3 -366999.309}
SPL {X  -159.990, Y  +656.991, Z    +0.000, E1  +350.742, E3 -367000.728}
SPL {X  -159.990, Y  +648.067, Z    +0.000, E1  +342.328, E3 -367004.457}
SPL {X  -159.990, Y  +620.451, Z    +0.000, E1  +325.419, E3 -367028.305}
SPL {X  -159.990, Y  +591.256, Z    +0.000, E1  +319.966, E3 -367074.798}
SPL {X  -159.990, Y  +586.740, Z    +0.000, E1  +319.956, E3 -367086.188}
SPL {X  -159.990, Y  +581.814, Z    +0.000, E1  +319.956, E3 -367098.628}
SPL {X  -159.990, Y  +577.274, Z    +0.000, E1  +319.964, E3 -367110.105}
SPL {X  -159.990, Y  +572.933, Z    +0.000, E1  +319.959, E3 -367121.047}
SPL {X  -159.990, Y  +568.504, Z    +0.000, E1  +319.956, E3 -367132.209}
SPL {X  -159.990, Y  +563.189, Z    +0.000, E1  +319.932, E3 -367145.583}
SPL {X  -159.990, Y  +557.707, Z    +0.000, E1  +319.949, E3 -367159.438}
SPL {X  -159.990, Y  +552.104, Z    +0.000, E1  +319.922, E3 -367173.513}
SPL {X  -159.990, Y  +545.912, Z    +0.000, E1  +319.929, E3 -367189.162}
SPL {X  -159.990, Y  +540.054, Z    +0.000, E1  +319.939, E3 -367203.990}
SPL {X  -159.990, Y  +533.683, Z    +0.000, E1  +319.916, E3 -367220.014}
SPL {X  -159.990, Y  +527.393, Z    +0.000, E1  +319.924, E3 -367235.887}
SPL {X  -159.990, Y  +522.533, Z    +0.000, E1  +319.951, E3 -367248.184}
SPL {X  -159.990, Y  +496.806, Z    +0.000, E1  +312.216, E3 -367258.392}
SPL {X  -159.990, Y  +490.245, Z    +0.000, E1  +312.831, E3 -367274.923}
SPL {X  -159.990, Y  +486.737, Z    +0.000, E1  +313.729, E3 -367286.929}
SPL {X  -159.990, Y  +483.955, Z    +0.000, E1  +314.316, E3 -367296.221}
SPL {X  -159.990, Y  +479.762, Z    +0.000, E1  +315.381, E3 -367311.612}
SPL {X  -159.990, Y  +475.871, Z    +0.000, E1  +316.362, E3 -367325.661}
SPL {X  -159.990, Y  +472.671, Z    +0.000, E1  +317.192, E3 -367337.964}
SPL {X  -159.990, Y  +468.809, Z    +0.000, E1  +318.343, E3 -367353.893}
SPL {X  -159.990, Y  +465.057, Z    +0.000, E1  +319.375, E3 -367369.051}
SPL {X  -159.990, Y  +461.409, Z    +0.000, E1  +319.848, E3 -367380.951}
SPL {X  -159.990, Y  +456.934, Z    +0.000, E1  +319.854, E3 -367392.227}
SPL {X  -159.990, Y  +452.940, Z    +0.000, E1  +319.854, E3 -367402.271}
SPL {X  -159.990, Y  +448.856, Z    +0.000, E1  +319.859, E3 -367412.554}
SPL {X  -159.990, Y  +444.973, Z    +0.000, E1  +319.856, E3 -367422.320}
SPL {X  -159.990, Y  +439.927, Z    +0.000, E1  +319.837, E3 -367434.976}
SPL {X  -159.990, Y  +435.246, Z    +0.000, E1  +319.853, E3 -367446.785}
SPL {X  -159.990, Y  +430.690, Z    +0.000, E1  +319.854, E3 -367458.247}
SPL {X  -159.990, Y  +426.145, Z    +0.000, E1  +319.853, E3 -367469.687}
SPL {X  -159.990, Y  +421.880, Z    +0.000, E1  +319.860, E3 -367480.420}
SPL {X  -159.990, Y  +416.246, Z    +0.000, E1  +319.819, E3 -367494.549}
SPL {X  -159.990, Y  +409.936, Z    +0.000, E1  +319.849, E3 -367510.486}
SPL {X  -159.990, Y  +404.988, Z    +0.000, E1  +319.861, E3 -367522.951}
SPL {X  -159.990, Y  +400.535, Z    +0.000, E1  +319.859, E3 -367534.149}
SPL {X  -159.990, Y  +396.024, Z    +0.000, E1  +319.860, E3 -367545.505}
SPL {X  -159.990, Y  +391.614, Z    +0.000, E1  +319.860, E3 -367556.599}
SPL {X  -159.990, Y  +387.212, Z    +0.000, E1  +319.859, E3 -367567.671}
SPL {X  -159.990, Y  +382.743, Z    +0.000, E1  +319.857, E3 -367578.913}
SPL {X  -159.925, Y  +377.946, Z    +0.000, E1  +319.864, E3 -367591.050}
SPL {X  -159.703, Y  +372.915, Z    +0.000, E1  +319.904, E3 -367603.949}
SPL {X  -159.358, Y  +368.290, Z    +0.000, E1  +319.961, E3 -367615.912}
SPL {X  -158.955, Y  +364.333, Z    +0.000, E1  +320.046, E3 -367626.314}
SPL {X  -158.482, Y  +360.589, Z    +0.000, E1  +320.125, E3 -367636.241}
SPL {X  -157.729, Y  +355.695, Z    +0.000, E1  +320.237, E3 -367649.313}
SPL {X  -156.893, Y  +351.173, Z    +0.000, E1  +320.410, E3 -367661.597}
SPL {X  -156.148, Y  +347.650, Z    +0.000, E1  +320.549, E3 -367671.242}
SPL {X  -155.268, Y  +343.918, Z    +0.000, E1  +320.696, E3 -367681.523}
SPL {X  -154.153, Y  +339.677, Z    +0.000, E1  +320.896, E3 -367693.330}
SPL {X  -152.885, Y  +335.352, Z    +0.000, E1  +321.114, E3 -367705.484}
SPL {X  -151.010, Y  +329.654, Z    +0.000, E1  +326.674, E3 -367765.700}
ENDSPLINE

SPLINE
SPL {X  -157.513, Y  +354.453, Z    +0.000, E1  +340.941, E3 -367811.735}
SPL {X  -159.408, Y  +368.861, Z    +0.000, E1  +348.865, E3 -367821.158}
SPL {X  -159.941, Y  +378.532, Z    +0.000, E1  +354.551, E3 -367824.763}
SPL {X  -159.990, Y  +383.966, Z    +0.000, E1  +358.149, E3 -367826.215}
SPL {X  -159.990, Y  +389.165, Z    +0.000, E1  +361.929, E3 -367827.417}
SPL {X  -159.990, Y  +396.368, Z    +0.000, E1  +368.359, E3 -367829.389}
SPL {X  -159.990, Y  +406.530, Z    +0.000, E1  +377.917, E3 -367833.771}
SPL {X  -159.990, Y  +429.014, Z    +0.000, E1  +392.438, E3 -367852.428}
SPL {X  -159.990, Y  +437.635, Z    +0.000, E1  +395.495, E3 -367862.660}
SPL {X  -159.990, Y  +460.330, Z    +0.000, E1  +398.908, E3 -367903.347}
SPL {X  -159.990, Y  +464.953, Z    +0.000, E1  +398.907, E3 -367915.506}
SPL {X  -159.990, Y  +469.353, Z    +0.000, E1  +398.902, E3 -367927.086}
SPL {X  -159.990, Y  +473.222, Z    +0.000, E1  +398.891, E3 -367937.295}
SPL {X  -159.990, Y  +477.957, Z    +0.000, E1  +398.922, E3 -367949.700}
SPL {X  -159.990, Y  +482.463, Z    +0.000, E1  +398.891, E3 -367961.587}
SPL {X  -159.990, Y  +486.996, Z    +0.000, E1  +398.928, E3 -367973.419}
SPL {X  -159.990, Y  +492.629, Z    +0.000, E1  +398.922, E3 -367988.226}
SPL {X  -159.990, Y  +497.431, Z    +0.000, E1  +398.905, E3 -368000.892}
SPL {X  -159.990, Y  +502.093, Z    +0.000, E1  +398.909, E3 -368013.167}
SPL {X  -159.990, Y  +507.821, Z    +0.000, E1  +398.930, E3 -368028.187}
SPL {X  -159.990, Y  +513.533, Z    +0.000, E1  +398.910, E3 -368043.246}
SPL {X  -159.990, Y  +519.462, Z    +0.000, E1  +398.933, E3 -368058.799}
SPL {X  -159.990, Y  +524.415, Z    +0.000, E1  +398.896, E3 -368071.863}
SPL {X  -159.990, Y  +528.627, Z    +0.000, E1  +398.910, E3 -368082.924}
SPL {X  -159.990, Y  +534.392, Z    +0.000, E1  +398.932, E3 -368098.054}
SPL {X  -159.990, Y  +540.299, Z    +0.000, E1  +398.912, E3 -368113.628}
SPL {X  -159.990, Y  +544.229, Z    +0.000, E1  +398.885, E3 -368124.002}
SPL {X  -159.990, Y  +549.483, Z    +0.000, E1  +398.950, E3 -368137.718}
SPL {X  -159.990, Y  +556.271, Z    +0.000, E1  +398.927, E3 -368155.588}
SPL {X  -159.990, Y  +561.696, Z    +0.000, E1  +398.912, E3 -368169.857}
SPL {X  -159.990, Y  +566.650, Z    +0.000, E1  +398.917, E3 -368182.871}
SPL {X  -159.990, Y  +571.814, Z    +0.000, E1  +398.914, E3 -368196.474}
SPL {X  -159.990, Y  +577.636, Z    +0.000, E1  +398.929, E3 -368211.771}
SPL {X  -159.990, Y  +583.167, Z    +0.000, E1  +398.906, E3 -368226.347}
SPL {X  -159.990, Y  +587.761, Z    +0.000, E1  +398.902, E3 -368238.431}
SPL {X  -159.990, Y  +592.962, Z    +0.000, E1  +398.925, E3 -368252.076}
SPL {X  -159.990, Y  +599.478, Z    +0.000, E1  +398.941, E3 -368269.186}
SPL {X  -159.990, Y  +606.904, Z    +0.000, E1  +398.953, E3 -368288.699}
SPL {X  -159.990, Y  +614.125, Z    +0.000, E1  +398.936, E3 -368307.711}
SPL {X  -159.990, Y  +619.061, Z    +0.000, E1  +398.894, E3 -368320.743}
SPL {X  -159.990, Y  +623.264, Z    +0.000, E1  +398.906, E3 -368331.792}
SPL {X  -159.990, Y  +628.669, Z    +0.000, E1  +398.928, E3 -368345.960}
SPL {X  -159.990, Y  +634.089, Z    +0.000, E1  +398.907, E3 -368360.236}
SPL {X  -159.990, Y  +638.639, Z    +0.000, E1  +398.904, E3 -368372.221}
SPL {X  -159.990, Y  +643.555, Z    +0.000, E1  +398.910, E3 -368385.141}
SPL {X  -159.990, Y  +649.380, Z    +0.000, E1  +398.930, E3 -368400.419}
SPL {X  -159.990, Y  +654.813, Z    +0.000, E1  +398.905, E3 -368414.743}
SPL {X  -159.990, Y  +658.715, Z    +0.000, E1  +398.892, E3 -368425.024}
SPL {X  -159.990, Y  +661.848, Z    +0.000, E1  +398.892, E3 -368433.263}
SPL {X  -159.990, Y  +665.703, Z    +0.000, E1  +398.903, E3 -368443.382}
SPL {X  -159.990, Y  +669.966, Z    +0.000, E1  +398.902, E3 -368454.589}
SPL {X  -159.954, Y  +674.895, Z    +0.000, E1  +398.910, E3 -368467.568}
SPL {X  -159.761, Y  +680.061, Z    +0.000, E1  +398.873, E3 -368481.348}
SPL {X  -159.443, Y  +684.716, Z    +0.000, E1  +398.815, E3 -368493.913}
SPL {X  -158.962, Y  +689.604, Z    +0.000, E1  +398.740, E3 -368507.282}
SPL {X  -158.139, Y  +695.766, Z    +0.000, E1  +398.623, E3 -368524.328}
SPL {X  -157.275, Y  +700.848, Z    +0.000, E1  +398.415, E3 -368538.680}
SPL {X  -156.506, Y  +704.705, Z    +0.000, E1  +398.294, E3 -368549.603}
SPL {X  -155.680, Y  +708.387, Z    +0.000, E1  +398.127, E3 -368560.174}
SPL {X  -154.586, Y  +712.730, Z    +0.000, E1  +397.967, E3 -368572.671}
SPL {X  -153.345, Y  +717.131, Z    +0.000, E1  +397.713, E3 -368585.555}
SPL {X  -151.080, Y  +724.146, Z    +0.000, E1  +393.201, E3 -368644.009}
ENDSPLINE

SPLINE
SPL {X  -157.921, Y  +697.149, Z    +0.000, E1  +377.701, E3 -368695.569}
SPL {X  -159.579, Y  +682.959, Z    +0.000, E1  +369.793, E3 -368703.518}
SPL {X  -159.938, Y  +675.561, Z    +0.000, E1  +365.399, E3 -368705.940}
SPL {X  -159.990, Y  +669.910, Z    +0.000, E1  +361.710, E3 -368707.231}
SPL {X  -159.990, Y  +665.465, Z    +0.000, E1  +358.378, E3 -368708.148}
SPL {X  -159.990, Y  +661.791, Z    +0.000, E1  +355.213, E3 -368708.986}
SPL {X  -159.990, Y  +656.991, Z    +0.000, E1  +350.742, E3 -368710.405}
SPL {X  -159.990, Y  +648.067, Z    +0.000, E1  +342.328, E3 -368714.135}
SPL {X  -159.990, Y  +624.891, Z    +0.000, E1  +327.004, E3 -368732.623}
SPL {X  -159.990, Y  +618.109, Z    +0.000, E1  +324.631, E3 -368740.799}
SPL {X  -159.990, Y  +591.256, Z    +0.000, E1  +319.966, E3 -368784.476}
SPL {X  -159.990, Y  +586.740, Z    +0.000, E1  +319.956, E3 -368795.866}
SPL {X  -159.990, Y  +581.814, Z    +0.000, E1  +319.956, E3 -368808.305}
SPL {X  -159.990, Y  +577.274, Z    +0.000, E1  +319.964, E3 -368819.783}
SPL {X  -159.990, Y  +572.933, Z    +0.000, E1  +319.959, E3 -368830.724}
SPL {X  -159.990, Y  +568.504, Z    +0.000, E1  +319.956, E3 -368841.887}
SPL {X  -159.990, Y  +564.427, Z    +0.000, E1  +319.959, E3 -368852.173}
SPL {X  -159.990, Y  +558.823, Z    +0.000, E1  +319.916, E3 -368866.252}
SPL {X  -159.990, Y  +553.571, Z    +0.000, E1  +319.954, E3 -368879.534}
SPL {X  -159.990, Y  +549.413, Z    +0.000, E1  +319.938, E3 -368890.000}
SPL {X  -159.990, Y  +544.924, Z    +0.000, E1  +319.955, E3 -368901.381}
SPL {X  -159.990, Y  +540.054, Z    +0.000, E1  +319.939, E3 -368913.667}
SPL {X  -159.990, Y  +533.683, Z    +0.000, E1  +319.916, E3 -368929.692}
SPL {X  -159.990, Y  +528.899, Z    +0.000, E1  +319.955, E3 -368941.808}
SPL {X  -159.990, Y  +523.984, Z    +0.000, E1  +319.922, E3 -368954.155}
SPL {X  -159.990, Y  +495.402, Z    +0.000, E1  +312.238, E3 -368971.085}
SPL {X  -159.990, Y  +488.437, Z    +0.000, E1  +313.241, E3 -368990.648}
SPL {X  -159.990, Y  +483.955, Z    +0.000, E1  +314.316, E3 -369005.899}
SPL {X  -159.990, Y  +480.580, Z    +0.000, E1  +315.242, E3 -369018.520}
SPL {X  -159.990, Y  +476.546, Z    +0.000, E1  +316.165, E3 -369032.815}
SPL {X  -159.990, Y  +473.377, Z    +0.000, E1  +316.953, E3 -369044.429}
SPL {X  -159.990, Y  +470.788, Z    +0.000, E1  +317.853, E3 -369055.843}
SPL {X  -159.990, Y  +467.944, Z    +0.000, E1  +318.635, E3 -369067.164}
SPL {X  -159.990, Y  +465.057, Z    +0.000, E1  +319.375, E3 -369078.729}
SPL {X  -159.990, Y  +461.409, Z    +0.000, E1  +319.848, E3 -369090.628}
SPL {X  -159.990, Y  +456.934, Z    +0.000, E1  +319.854, E3 -369101.904}
SPL {X  -159.990, Y  +452.940, Z    +0.000, E1  +319.854, E3 -369111.949}
SPL {X  -159.990, Y  +448.856, Z    +0.000, E1  +319.859, E3 -369122.232}
SPL {X  -159.990, Y  +444.973, Z    +0.000, E1  +319.856, E3 -369131.997}
SPL {X  -159.990, Y  +439.927, Z    +0.000, E1  +319.837, E3 -369144.654}
SPL {X  -159.990, Y  +435.246, Z    +0.000, E1  +319.853, E3 -369156.463}
SPL {X  -159.990, Y  +430.690, Z    +0.000, E1  +319.854, E3 -369167.925}
SPL {X  -159.990, Y  +426.145, Z    +0.000, E1  +319.853, E3 -369179.365}
SPL {X  -159.990, Y  +421.880, Z    +0.000, E1  +319.860, E3 -369190.097}
SPL {X  -159.990, Y  +416.246, Z    +0.000, E1  +319.819, E3 -369204.226}
SPL {X  -159.990, Y  +409.936, Z    +0.000, E1  +319.849, E3 -369220.163}
SPL {X  -159.990, Y  +404.988, Z    +0.000, E1  +319.861, E3 -369232.629}
SPL {X  -159.990, Y  +400.535, Z    +0.000, E1  +319.859, E3 -369243.827}
SPL {X  -159.990, Y  +396.024, Z    +0.000, E1  +319.860, E3 -369255.183}
SPL {X  -159.990, Y  +391.614, Z    +0.000, E1  +319.860, E3 -369266.276}
SPL {X  -159.990, Y  +387.212, Z    +0.000, E1  +319.859, E3 -369277.348}
SPL {X  -159.990, Y  +382.743, Z    +0.000, E1  +319.857, E3 -369288.590}
SPL {X  -159.925, Y  +377.946, Z    +0.000, E1  +319.864, E3 -369300.727}
SPL {X  -159.703, Y  +372.915, Z    +0.000, E1  +319.904, E3 -369313.627}
SPL {X  -159.358, Y  +368.290, Z    +0.000, E1  +319.961, E3 -369325.589}
SPL {X  -158.955, Y  +364.333, Z    +0.000, E1  +320.046, E3 -369335.992}
SPL {X  -158.482, Y  +360.589, Z    +0.000, E1  +320.125, E3 -369345.918}
SPL {X  -157.729, Y  +355.695, Z    +0.000, E1  +320.237, E3 -369358.991}
SPL {X  -156.893, Y  +351.173, Z    +0.000, E1  +320.410, E3 -369371.274}
SPL {X  -156.148, Y  +347.650, Z    +0.000, E1  +320.549, E3 -369380.920}
SPL {X  -155.268, Y  +343.918, Z    +0.000, E1  +320.696, E3 -369391.201}
SPL {X  -154.153, Y  +339.677, Z    +0.000, E1  +320.896, E3 -369403.008}
SPL {X  -152.885, Y  +335.352, Z    +0.000, E1  +321.114, E3 -369415.162}
SPL {X  -151.010, Y  +329.654, Z    +0.000, E1  +326.674, E3 -369475.378}
ENDSPLINE

SPLINE
SPL {X  -157.513, Y  +354.453, Z    +0.000, E1  +340.941, E3 -369521.412}
SPL {X  -159.408, Y  +368.861, Z    +0.000, E1  +348.865, E3 -369530.835}
SPL {X  -159.941, Y  +378.532, Z    +0.000, E1  +354.551, E3 -369534.441}
SPL {X  -159.990, Y  +383.966, Z    +0.000, E1  +358.149, E3 -369535.892}
SPL {X  -159.990, Y  +388.001, Z    +0.000, E1  +361.086, E3 -369536.828}
SPL {X  -159.990, Y  +392.647, Z    +0.000, E1  +364.974, E3 -369537.966}
SPL {X  -159.990, Y  +397.943, Z    +0.000, E1  +369.963, E3 -369539.551}
SPL {X  -159.990, Y  +407.689, Z    +0.000, E1  +378.860, E3 -369544.205}
SPL {X  -159.990, Y  +434.822, Z    +0.000, E1  +394.625, E3 -369568.749}
SPL {X  -159.990, Y  +460.330, Z    +0.000, E1  +398.908, E3 -369613.025}
SPL {X  -159.990, Y  +464.953, Z    +0.000, E1  +398.907, E3 -369625.183}
SPL {X  -159.990, Y  +469.353, Z    +0.000, E1  +398.902, E3 -369636.763}
SPL {X  -159.990, Y  +473.222, Z    +0.000, E1  +398.891, E3 -369646.972}
SPL {X  -159.990, Y  +477.957, Z    +0.000, E1  +398.922, E3 -369659.377}
SPL {X  -159.990, Y  +482.463, Z    +0.000, E1  +398.891, E3 -369671.265}
SPL {X  -159.990, Y  +486.996, Z    +0.000, E1  +398.928, E3 -369683.097}
SPL {X  -159.990, Y  +492.629, Z    +0.000, E1  +398.922, E3 -369697.903}
SPL {X  -159.990, Y  +497.431, Z    +0.000, E1  +398.905, E3 -369710.570}
SPL {X  -159.990, Y  +502.093, Z    +0.000, E1  +398.909, E3 -369722.844}
SPL {X  -159.990, Y  +507.821, Z    +0.000, E1  +398.930, E3 -369737.864}
SPL {X  -159.990, Y  +513.533, Z    +0.000, E1  +398.910, E3 -369752.924}
SPL {X  -159.990, Y  +519.462, Z    +0.000, E1  +398.933, E3 -369768.476}
SPL {X  -159.990, Y  +524.415, Z    +0.000, E1  +398.896, E3 -369781.541}
SPL {X  -159.990, Y  +528.627, Z    +0.000, E1  +398.910, E3 -369792.601}
SPL {X  -159.990, Y  +534.392, Z    +0.000, E1  +398.932, E3 -369807.731}
SPL {X  -159.990, Y  +540.299, Z    +0.000, E1  +398.912, E3 -369823.306}
SPL {X  -159.990, Y  +545.676, Z    +0.000, E1  +398.913, E3 -369837.443}
SPL {X  -159.990, Y  +550.777, Z    +0.000, E1  +398.906, E3 -369850.863}
SPL {X  -159.990, Y  +556.271, Z    +0.000, E1  +398.927, E3 -369865.265}
SPL {X  -159.990, Y  +561.696, Z    +0.000, E1  +398.912, E3 -369879.535}
SPL {X  -159.990, Y  +566.650, Z    +0.000, E1  +398.917, E3 -369892.548}
SPL {X  -159.990, Y  +571.814, Z    +0.000, E1  +398.914, E3 -369906.151}
SPL {X  -159.990, Y  +577.636, Z    +0.000, E1  +398.929, E3 -369921.448}
SPL {X  -159.990, Y  +583.167, Z    +0.000, E1  +398.906, E3 -369936.024}
SPL {X  -159.990, Y  +587.761, Z    +0.000, E1  +398.902, E3 -369948.109}
SPL {X  -159.990, Y  +592.962, Z    +0.000, E1  +398.925, E3 -369961.753}
SPL {X  -159.990, Y  +597.767, Z    +0.000, E1  +398.897, E3 -369974.428}
SPL {X  -159.990, Y  +602.727, Z    +0.000, E1  +398.920, E3 -369987.439}
SPL {X  -159.990, Y  +608.112, Z    +0.000, E1  +398.911, E3 -370001.614}
SPL {X  -159.990, Y  +613.039, Z    +0.000, E1  +398.906, E3 -370014.576}
SPL {X  -159.990, Y  +618.087, Z    +0.000, E1  +398.915, E3 -370027.835}
SPL {X  -159.990, Y  +623.264, Z    +0.000, E1  +398.906, E3 -370041.469}
SPL {X  -159.990, Y  +628.669, Z    +0.000, E1  +398.928, E3 -370055.637}
SPL {X  -159.990, Y  +634.089, Z    +0.000, E1  +398.907, E3 -370069.913}
SPL {X  -159.990, Y  +638.639, Z    +0.000, E1  +398.904, E3 -370081.899}
SPL {X  -159.990, Y  +643.555, Z    +0.000, E1  +398.910, E3 -370094.819}
SPL {X  -159.990, Y  +649.380, Z    +0.000, E1  +398.930, E3 -370110.096}
SPL {X  -159.990, Y  +654.813, Z    +0.000, E1  +398.905, E3 -370124.421}
SPL {X  -159.990, Y  +660.353, Z    +0.000, E1  +398.930, E3 -370138.952}
SPL {X  -159.990, Y  +665.703, Z    +0.000, E1  +398.903, E3 -370153.060}
SPL {X  -159.990, Y  +669.966, Z    +0.000, E1  +398.902, E3 -370164.266}
SPL {X  -159.954, Y  +674.895, Z    +0.000, E1  +398.910, E3 -370177.246}
SPL {X  -159.761, Y  +680.061, Z    +0.000, E1  +398.873, E3 -370191.025}
SPL {X  -159.443, Y  +684.716, Z    +0.000, E1  +398.815, E3 -370203.590}
SPL {X  -158.962, Y  +689.604, Z    +0.000, E1  +398.740, E3 -370216.959}
SPL {X  -158.318, Y  +694.567, Z    +0.000, E1  +398.614, E3 -370230.720}
SPL {X  -157.472, Y  +699.775, Z    +0.000, E1  +398.483, E3 -370245.280}
SPL {X  -156.506, Y  +704.705, Z    +0.000, E1  +398.294, E3 -370259.280}
SPL {X  -155.680, Y  +708.387, Z    +0.000, E1  +398.127, E3 -370269.851}
SPL {X  -154.586, Y  +712.730, Z    +0.000, E1  +397.967, E3 -370282.348}
SPL {X  -153.345, Y  +717.131, Z    +0.000, E1  +397.713, E3 -370295.232}
SPL {X  -151.080, Y  +724.146, Z    +0.000, E1  +393.201, E3 -370353.686}
ENDSPLINE

SPLINE
SPL {X  -157.921, Y  +697.149, Z    +0.000, E1  +377.701, E3 -370405.247}
SPL {X  -159.579, Y  +682.959, Z    +0.000, E1  +369.793, E3 -370413.195}
SPL {X  -159.938, Y  +675.561, Z    +0.000, E1  +365.399, E3 -370415.617}
SPL {X  -159.990, Y  +669.910, Z    +0.000, E1  +361.710, E3 -370416.908}
SPL {X  -159.990, Y  +665.465, Z    +0.000, E1  +358.378, E3 -370417.826}
SPL {X  -159.990, Y  +661.791, Z    +0.000, E1  +355.213, E3 -370418.663}
SPL {X  -159.990, Y  +656.991, Z    +0.000, E1  +350.742, E3 -370420.083}
SPL {X  -159.990, Y  +648.067, Z    +0.000, E1  +342.328, E3 -370423.812}
SPL {X  -159.990, Y  +620.451, Z    +0.000, E1  +325.419, E3 -370447.659}
SPL {X  -159.990, Y  +591.256, Z    +0.000, E1  +319.966, E3 -370494.153}
SPL {X  -159.990, Y  +586.740, Z    +0.000, E1  +319.956, E3 -370505.543}
SPL {X  -159.990, Y  +581.814, Z    +0.000, E1  +319.956, E3 -370517.983}
SPL {X  -159.990, Y  +577.274, Z    +0.000, E1  +319.964, E3 -370529.460}
SPL {X  -159.990, Y  +572.933, Z    +0.000, E1  +319.959, E3 -370540.401}
SPL {X  -159.990, Y  +568.504, Z    +0.000, E1  +319.956, E3 -370551.564}
SPL {X  -159.990, Y  +563.189, Z    +0.000, E1  +319.932, E3 -370564.938}
SPL {X  -159.990, Y  +557.707, Z    +0.000, E1  +319.949, E3 -370578.793}
SPL {X  -159.990, Y  +552.104, Z    +0.000, E1  +319.922, E3 -370592.868}
SPL {X  -159.990, Y  +545.912, Z    +0.000, E1  +319.929, E3 -370608.517}
SPL {X  -159.990, Y  +540.054, Z    +0.000, E1  +319.939, E3 -370623.344}
SPL {X  -159.990, Y  +533.683, Z    +0.000, E1  +319.916, E3 -370639.369}
SPL {X  -159.990, Y  +527.393, Z    +0.000, E1  +319.924, E3 -370655.242}
SPL {X  -159.990, Y  +522.533, Z    +0.000, E1  +319.951, E3 -370667.539}
SPL {X  -159.990, Y  +496.806, Z    +0.000, E1  +312.216, E3 -370677.747}
SPL {X  -159.990, Y  +490.245, Z    +0.000, E1  +312.831, E3 -370694.278}
SPL {X  -159.990, Y  +486.737, Z    +0.000, E1  +313.729, E3 -370706.284}
SPL {X  -159.990, Y  +483.955, Z    +0.000, E1  +314.316, E3 -370715.576}
SPL {X  -159.990, Y  +479.762, Z    +0.000, E1  +315.381, E3 -370730.967}
SPL {X  -159.990, Y  +475.871, Z    +0.000, E1  +316.362, E3 -370745.016}
SPL {X  -159.990, Y  +472.671, Z    +0.000, E1  +317.192, E3 -370757.319}
SPL {X  -159.990, Y  +468.809, Z    +0.000, E1  +318.343, E3 -370773.248}
SPL {X  -159.990, Y  +465.057, Z    +0.000, E1  +319.375, E3 -370788.406}
SPL {X  -159.990, Y  +461.409, Z    +0.000, E1  +319.848, E3 -370800.306}
SPL {X  -159.990, Y  +456.934, Z    +0.000, E1  +319.854, E3 -370811.581}
SPL {X  -159.990, Y  +452.940, Z    +0.000, E1  +319.854, E3 -370821.626}
SPL {X  -159.990, Y  +448.856, Z    +0.000, E1  +319.859, E3 -370831.909}
SPL {X  -159.990, Y  +444.973, Z    +0.000, E1  +319.856, E3 -370841.675}
SPL {X  -159.990, Y  +439.927, Z    +0.000, E1  +319.837, E3 -370854.331}
SPL {X  -159.990, Y  +435.246, Z    +0.000, E1  +319.853, E3 -370866.140}
SPL {X  -159.990, Y  +430.690, Z    +0.000, E1  +319.854, E3 -370877.602}
SPL {X  -159.990, Y  +426.145, Z    +0.000, E1  +319.853, E3 -370889.042}
SPL {X  -159.990, Y  +421.880, Z    +0.000, E1  +319.860, E3 -370899.775}
SPL {X  -159.990, Y  +416.246, Z    +0.000, E1  +319.819, E3 -370913.904}
SPL {X  -159.990, Y  +409.936, Z    +0.000, E1  +319.849, E3 -370929.840}
SPL {X  -159.990, Y  +404.988, Z    +0.000, E1  +319.861, E3 -370942.306}
SPL {X  -159.990, Y  +400.535, Z    +0.000, E1  +319.859, E3 -370953.504}
SPL {X  -159.990, Y  +396.024, Z    +0.000, E1  +319.860, E3 -370964.860}
SPL {X  -159.990, Y  +391.614, Z    +0.000, E1  +319.860, E3 -370975.954}
SPL {X  -159.990, Y  +387.212, Z    +0.000, E1  +319.859, E3 -370987.026}
SPL {X  -159.990, Y  +382.743, Z    +0.000, E1  +319.857, E3 -370998.267}
SPL {X  -159.925, Y  +377.946, Z    +0.000, E1  +319.864, E3 -371010.404}
SPL {X  -159.703, Y  +372.915, Z    +0.000, E1  +319.904, E3 -371023.304}
SPL {X  -159.358, Y  +368.290, Z    +0.000, E1  +319.961, E3 -371035.267}
SPL {X  -158.955, Y  +364.333, Z    +0.000, E1  +320.046, E3 -371045.669}
SPL {X  -158.482, Y  +360.589, Z    +0.000, E1  +320.125, E3 -371055.595}
SPL {X  -157.729, Y  +355.695, Z    +0.000, E1  +320.237, E3 -371068.668}
SPL {X  -156.893, Y  +351.173, Z    +0.000, E1  +320.410, E3 -371080.951}
SPL {X  -156.148, Y  +347.650, Z    +0.000, E1  +320.549, E3 -371090.597}
SPL {X  -155.268, Y  +343.918, Z    +0.000, E1  +320.696, E3 -371100.878}
SPL {X  -154.153, Y  +339.677, Z    +0.000, E1  +320.896, E3 -371112.685}
SPL {X  -152.885, Y  +335.352, Z    +0.000, E1  +321.114, E3 -371124.839}
SPL {X  -151.010, Y  +329.654, Z    +0.000, E1  +326.674, E3 -371185.055}
ENDSPLINE

SPLINE
SPL {X  -157.513, Y  +354.453, Z    +0.000, E1  +340.941, E3 -371231.090}
SPL {X  -159.408, Y  +368.861, Z    +0.000, E1  +348.865, E3 -371240.512}
SPL {X  -159.941, Y  +378.532, Z    +0.000, E1  +354.551, E3 -371244.118}
SPL {X  -159.990, Y  +383.966, Z    +0.000, E1  +358.149, E3 -371245.570}
SPL {X  -159.990, Y  +389.165, Z    +0.000, E1  +361.929, E3 -371246.772}
SPL {X  -159.990, Y  +396.368, Z    +0.000, E1  +368.359, E3 -371248.744}
SPL {X  -159.990, Y  +406.530, Z    +0.000, E1  +377.917, E3 -371253.126}
SPL {X  -159.990, Y  +429.014, Z    +0.000, E1  +392.438, E3 -371271.782}
SPL {X  -159.990, Y  +437.635, Z    +0.000, E1  +395.495, E3 -371282.015}
SPL {X  -159.990, Y  +460.330, Z    +0.000, E1  +398.908, E3 -371322.702}
SPL {X  -159.990, Y  +464.953, Z    +0.000, E1  +398.907, E3 -371334.860}
SPL {X  -159.990, Y  +469.353, Z    +0.000, E1  +398.902, E3 -371346.441}
SPL {X  -159.990, Y  +473.222, Z    +0.000, E1  +398.891, E3 -371356.649}
SPL {X  -159.990, Y  +477.957, Z    +0.000, E1  +398.922, E3 -371369.054}
SPL {X  -159.990, Y  +482.463, Z    +0.000, E1  +398.891, E3 -371380.942}
SPL {X  -159.990, Y  +486.996, Z    +0.000, E1  +398.928, E3 -371392.774}
SPL {X  -159.990, Y  +492.629, Z    +0.000, E1  +398.922, E3 -371407.581}
SPL {X  -159.990, Y  +497.431, Z    +0.000, E1  +398.905, E3 -371420.247}
SPL {X  -159.990, Y  +502.093, Z    +0.000, E1  +398.909, E3 -371432.522}
SPL {X  -159.990, Y  +507.821, Z    +0.000, E1  +398.930, E3 -371447.542}
SPL {X  -159.990, Y  +513.533, Z    +0.000, E1  +398.910, E3 -371462.601}
SPL {X  -159.990, Y  +519.462, Z    +0.000, E1  +398.933, E3 -371478.154}
SPL {X  -159.990, Y  +524.415, Z    +0.000, E1  +398.896, E3 -371491.218}
SPL {X  -159.990, Y  +528.627, Z    +0.000, E1  +398.910, E3 -371502.278}
SPL {X  -159.990, Y  +534.392, Z    +0.000, E1  +398.932, E3 -371517.409}
SPL {X  -159.990, Y  +540.299, Z    +0.000, E1  +398.912, E3 -371532.983}
SPL {X  -159.990, Y  +544.229, Z    +0.000, E1  +398.885, E3 -371543.357}
SPL {X  -159.990, Y  +549.483, Z    +0.000, E1  +398.950, E3 -371557.073}
SPL {X  -159.990, Y  +556.271, Z    +0.000, E1  +398.927, E3 -371574.943}
SPL {X  -159.990, Y  +561.696, Z    +0.000, E1  +398.912, E3 -371589.212}
SPL {X  -159.990, Y  +566.650, Z    +0.000, E1  +398.917, E3 -371602.226}
SPL {X  -159.990, Y  +571.814, Z    +0.000, E1  +398.914, E3 -371615.828}
SPL {X  -159.990, Y  +577.636, Z    +0.000, E1  +398.929, E3 -371631.126}
SPL {X  -159.990, Y  +583.167, Z    +0.000, E1  +398.906, E3 -371645.701}
SPL {X  -159.990, Y  +587.761, Z    +0.000, E1  +398.902, E3 -371657.786}
SPL {X  -159.990, Y  +592.962, Z    +0.000, E1  +398.925, E3 -371671.430}
SPL {X  -159.990, Y  +599.478, Z    +0.000, E1  +398.941, E3 -371688.541}
SPL {X  -159.990, Y  +606.904, Z    +0.000, E1  +398.953, E3 -371708.054}
SPL {X  -159.990, Y  +614.125, Z    +0.000, E1  +398.936, E3 -371727.066}
SPL {X  -159.990, Y  +619.061, Z    +0.000, E1  +398.894, E3 -371740.098}
SPL {X  -159.990, Y  +623.264, Z    +0.000, E1  +398.906, E3 -371751.147}
SPL {X  -159.990, Y  +628.669, Z    +0.000, E1  +398.928, E3 -371765.315}
SPL {X  -159.990, Y  +634.089, Z    +0.000, E1  +398.907, E3 -371779.591}
SPL {X  -159.990, Y  +638.639, Z    +0.000, E1  +398.904, E3 -371791.576}
SPL {X  -159.990, Y  +643.555, Z    +0.000, E1  +398.910, E3 -371804.496}
SPL {X  -159.990, Y  +649.380, Z    +0.000, E1  +398.930, E3 -371819.774}
SPL {X  -159.990, Y  +654.813, Z    +0.000, E1  +398.905, E3 -371834.098}
SPL {X  -159.990, Y  +658.715, Z    +0.000, E1  +398.892, E3 -371844.379}
SPL {X  -159.990, Y  +661.848, Z    +0.000, E1  +398.892, E3 -371852.618}
SPL {X  -159.990, Y  +665.703, Z    +0.000, E1  +398.903, E3 -371862.737}
SPL {X  -159.990, Y  +669.966, Z    +0.000, E1  +398.902, E3 -371873.944}
SPL {X  -159.954, Y  +674.895, Z    +0.000, E1  +398.910, E3 -371886.923}
SPL {X  -159.761, Y  +680.061, Z    +0.000, E1  +398.873, E3 -371900.702}
SPL {X  -159.443, Y  +684.716, Z    +0.000, E1  +398.815, E3 -371913.267}
SPL {X  -158.962, Y  +689.604, Z    +0.000, E1  +398.740, E3 -371926.637}
SPL {X  -158.139, Y  +695.766, Z    +0.000, E1  +398.623, E3 -371943.682}
SPL {X  -157.275, Y  +700.848, Z    +0.000, E1  +398.415, E3 -371958.034}
SPL {X  -156.506, Y  +704.705, Z    +0.000, E1  +398.294, E3 -371968.958}
SPL {X  -155.680, Y  +708.387, Z    +0.000, E1  +398.127, E3 -371979.529}
SPL {X  -154.586, Y  +712.730, Z    +0.000, E1  +397.967, E3 -371992.026}
SPL {X  -153.345, Y  +717.131, Z    +0.000, E1  +397.713, E3 -372004.910}
SPL {X  -151.080, Y  +724.146, Z    +0.000, E1  +393.201, E3 -372063.363}
ENDSPLINE

SPLINE
SPL {X  -157.921, Y  +697.149, Z    +0.000, E1  +377.701, E3 -372114.924}
SPL {X  -159.579, Y  +682.959, Z    +0.000, E1  +369.793, E3 -372122.873}
SPL {X  -159.938, Y  +675.561, Z    +0.000, E1  +365.399, E3 -372125.295}
SPL {X  -159.990, Y  +669.910, Z    +0.000, E1  +361.710, E3 -372126.586}
SPL {X  -159.990, Y  +665.465, Z    +0.000, E1  +358.378, E3 -372127.503}
SPL {X  -159.990, Y  +661.791, Z    +0.000, E1  +355.213, E3 -372128.341}
SPL {X  -159.990, Y  +656.991, Z    +0.000, E1  +350.742, E3 -372129.760}
SPL {X  -159.990, Y  +648.067, Z    +0.000, E1  +342.328, E3 -372133.490}
SPL {X  -159.990, Y  +624.891, Z    +0.000, E1  +327.004, E3 -372151.978}
SPL {X  -159.990, Y  +618.109, Z    +0.000, E1  +324.631, E3 -372160.154}
SPL {X  -159.990, Y  +591.256, Z    +0.000, E1  +319.966, E3 -372203.830}
SPL {X  -159.990, Y  +586.740, Z    +0.000, E1  +319.956, E3 -372215.221}
SPL {X  -159.990, Y  +581.814, Z    +0.000, E1  +319.956, E3 -372227.660}
SPL {X  -159.990, Y  +577.274, Z    +0.000, E1  +319.964, E3 -372239.138}
SPL {X  -159.990, Y  +572.933, Z    +0.000, E1  +319.959, E3 -372250.079}
SPL {X  -159.990, Y  +568.504, Z    +0.000, E1  +319.956, E3 -372261.241}
SPL {X  -159.990, Y  +563.189, Z    +0.000, E1  +319.932, E3 -372274.615}
SPL {X  -159.990, Y  +557.707, Z    +0.000, E1  +319.949, E3 -372288.470}
SPL {X  -159.990, Y  +552.104, Z    +0.000, E1  +319.922, E3 -372302.545}
SPL {X  -159.990, Y  +545.912, Z    +0.000, E1  +319.929, E3 -372318.195}
SPL {X  -159.990, Y  +541.567, Z    +0.000, E1  +319.969, E3 -372329.249}
SPL {X  -159.990, Y  +537.213, Z    +0.000, E1  +319.937, E3 -372340.185}
SPL {X  -159.990, Y  +532.291, Z    +0.000, E1  +319.951, E3 -372352.610}
SPL {X  -159.990, Y  +528.899, Z    +0.000, E1  +319.955, E3 -372361.163}
SPL {X  -159.990, Y  +523.984, Z    +0.000, E1  +319.922, E3 -372373.510}
SPL {X  -159.990, Y  +495.402, Z    +0.000, E1  +312.238, E3 -372390.440}
SPL {X  -159.990, Y  +489.464, Z    +0.000, E1  +313.059, E3 -372406.655}
SPL {X  -159.990, Y  +484.831, Z    +0.000, E1  +314.066, E3 -372422.188}
SPL {X  -159.990, Y  +479.762, Z    +0.000, E1  +315.381, E3 -372440.645}
SPL {X  -159.990, Y  +475.871, Z    +0.000, E1  +316.362, E3 -372454.693}
SPL {X  -159.990, Y  +472.671, Z    +0.000, E1  +317.192, E3 -372466.997}
SPL {X  -159.990, Y  +468.809, Z    +0.000, E1  +318.343, E3 -372482.925}
SPL {X  -159.990, Y  +465.057, Z    +0.000, E1  +319.375, E3 -372498.084}
SPL {X  -159.990, Y  +461.409, Z    +0.000, E1  +319.848, E3 -372509.983}
SPL {X  -159.990, Y  +456.934, Z    +0.000, E1  +319.854, E3 -372521.259}
SPL {X  -159.990, Y  +452.940, Z    +0.000, E1  +319.854, E3 -372531.303}
SPL {X  -159.990, Y  +448.856, Z    +0.000, E1  +319.859, E3 -372541.587}
SPL {X  -159.990, Y  +444.973, Z    +0.000, E1  +319.856, E3 -372551.352}
SPL {X  -159.990, Y  +439.927, Z    +0.000, E1  +319.837, E3 -372564.009}
SPL {X  -159.990, Y  +435.246, Z    +0.000, E1  +319.853, E3 -372575.818}
SPL {X  -159.990, Y  +430.690, Z    +0.000, E1  +319.854, E3 -372587.280}
SPL {X  -159.990, Y  +426.145, Z    +0.000, E1  +319.853, E3 -372598.719}
SPL {X  -159.990, Y  +421.880, Z    +0.000, E1  +319.860, E3 -372609.452}
SPL {X  -159.990, Y  +417.572, Z    +0.000, E1  +319.852, E3 -372620.279}
SPL {X  -159.990, Y  +412.619, Z    +0.000, E1  +319.850, E3 -372632.770}
SPL {X  -159.990, Y  +406.264, Z    +0.000, E1  +319.825, E3 -372648.719}
SPL {X  -159.990, Y  +400.535, Z    +0.000, E1  +319.859, E3 -372663.182}
SPL {X  -159.990, Y  +396.024, Z    +0.000, E1  +319.860, E3 -372674.538}
SPL {X  -159.990, Y  +391.614, Z    +0.000, E1  +319.860, E3 -372685.631}
SPL {X  -159.990, Y  +387.212, Z    +0.000, E1  +319.859, E3 -372696.703}
SPL {X  -159.990, Y  +382.743, Z    +0.000, E1  +319.857, E3 -372707.945}
SPL {X  -159.925, Y  +377.946, Z    +0.000, E1  +319.864, E3 -372720.082}
SPL {X  -159.703, Y  +372.915, Z    +0.000, E1  +319.904, E3 -372732.982}
SPL {X  -159.358, Y  +368.290, Z    +0.000, E1  +319.961, E3 -372744.944}
SPL {X  -158.955, Y  +364.333, Z    +0.000, E1  +320.046, E3 -372755.347}
SPL {X  -158.482, Y  +360.589, Z    +0.000, E1  +320.125, E3 -372765.273}
SPL {X  -157.729, Y  +355.695, Z    +0.000, E1  +320.237, E3 -372778.345}
SPL {X  -156.893, Y  +351.173, Z    +0.000, E1  +320.410, E3 -372790.629}
SPL {X  -156.148, Y  +347.650, Z    +0.000, E1  +320.549, E3 -372800.275}
SPL {X  -155.268, Y  +343.918, Z    +0.000, E1  +320.696, E3 -372810.555}
SPL {X  -154.153, Y  +339.677, Z    +0.000, E1  +320.896, E3 -372822.362}
SPL {X  -152.885, Y  +335.352, Z    +0.000, E1  +321.114, E3 -372834.517}
SPL {X  -151.010, Y  +329.654, Z    +0.000, E1  +326.674, E3 -372894.733}
ENDSPLINE

SPLINE
SPL {X  -157.513, Y  +354.453, Z    +0.000, E1  +340.941, E3 -372940.767}
SPL {X  -159.408, Y  +368.861, Z    +0.000, E1  +348.865, E3 -372950.190}
SPL {X  -159.941, Y  +378.532, Z    +0.000, E1  +354.551, E3 -372953.795}
SPL {X  -159.990, Y  +383.966, Z    +0.000, E1  +358.149, E3 -372955.247}
SPL {X  -159.990, Y  +389.165, Z    +0.000, E1  +361.929, E3 -372956.449}
SPL {X  -159.990, Y  +396.368, Z    +0.000, E1  +368.359, E3 -372958.421}
SPL {X  -159.990, Y  +407.689, Z    +0.000, E1  +378.860, E3 -372963.560}
SPL {X  -159.990, Y  +434.822, Z    +0.000, E1  +394.625, E3 -372988.104}
SPL {X  -159.990, Y  +460.330, Z    +0.000, E1  +398.908, E3 -373032.379}
SPL {X  -159.990, Y  +464.953, Z    +0.000, E1  +398.907, E3 -373044.538}
SPL {X  -159.990, Y  +469.353, Z    +0.000, E1  +398.902, E3 -373056.118}
SPL {X  -159.990, Y  +475.034, Z    +0.000, E1  +398.936, E3 -373071.033}
SPL {X  -159.990, Y  +481.308, Z    +0.000, E1  +398.917, E3 -373087.544}
SPL {X  -159.990, Y  +485.396, Z    +0.000, E1  +398.893, E3 -373098.303}
SPL {X  -159.990, Y  +489.893, Z    +0.000, E1  +398.930, E3 -373110.059}
SPL {X  -159.990, Y  +496.271, Z    +0.000, E1  +398.942, E3 -373126.815}
SPL {X  -159.990, Y  +502.093, Z    +0.000, E1  +398.909, E3 -373142.199}
SPL {X  -159.990, Y  +506.629, Z    +0.000, E1  +398.900, E3 -373154.131}
SPL {X  -159.990, Y  +512.483, Z    +0.000, E1  +398.947, E3 -373169.460}
SPL {X  -159.990, Y  +518.435, Z    +0.000, E1  +398.905, E3 -373185.174}
SPL {X  -159.990, Y  +523.478, Z    +0.000, E1  +398.918, E3 -373198.402}
SPL {X  -159.990, Y  +528.627, Z    +0.000, E1  +398.910, E3 -373211.956}
SPL {X  -159.990, Y  +533.053, Z    +0.000, E1  +398.899, E3 -373223.614}
SPL {X  -159.990, Y  +537.174, Z    +0.000, E1  +398.910, E3 -373234.428}
SPL {X  -159.990, Y  +542.636, Z    +0.000, E1  +398.920, E3 -373248.796}
SPL {X  -159.990, Y  +549.483, Z    +0.000, E1  +398.950, E3 -373266.751}
SPL {X  -159.990, Y  +554.638, Z    +0.000, E1  +398.890, E3 -373280.388}
SPL {X  -159.990, Y  +557.678, Z    +0.000, E1  +398.893, E3 -373288.364}
SPL {X  -159.990, Y  +561.696, Z    +0.000, E1  +398.912, E3 -373298.889}
SPL {X  -159.990, Y  +566.650, Z    +0.000, E1  +398.917, E3 -373311.903}
SPL {X  -159.990, Y  +571.814, Z    +0.000, E1  +398.914, E3 -373325.506}
SPL {X  -159.990, Y  +577.636, Z    +0.000, E1  +398.929, E3 -373340.803}
SPL {X  -159.990, Y  +583.167, Z    +0.000, E1  +398.906, E3 -373355.379}
SPL {X  -159.990, Y  +587.761, Z    +0.000, E1  +398.902, E3 -373367.464}
SPL {X  -159.990, Y  +592.962, Z    +0.000, E1  +398.925, E3 -373381.108}
SPL {X  -159.990, Y  +597.767, Z    +0.000, E1  +398.897, E3 -373393.783}
SPL {X  -159.990, Y  +602.727, Z    +0.000, E1  +398.920, E3 -373406.794}
SPL {X  -159.990, Y  +608.112, Z    +0.000, E1  +398.911, E3 -373420.968}
SPL {X  -159.990, Y  +613.039, Z    +0.000, E1  +398.906, E3 -373433.931}
SPL {X  -159.990, Y  +618.087, Z    +0.000, E1  +398.915, E3 -373447.190}
SPL {X  -159.990, Y  +623.264, Z    +0.000, E1  +398.906, E3 -373460.824}
SPL {X  -159.990, Y  +628.669, Z    +0.000, E1  +398.928, E3 -373474.992}
SPL {X  -159.990, Y  +634.089, Z    +0.000, E1  +398.907, E3 -373489.268}
SPL {X  -159.990, Y  +638.639, Z    +0.000, E1  +398.904, E3 -373501.254}
SPL {X  -159.990, Y  +644.750, Z    +0.000, E1  +398.946, E3 -373517.259}
SPL {X  -159.990, Y  +650.458, Z    +0.000, E1  +398.900, E3 -373532.331}
SPL {X  -159.990, Y  +654.813, Z    +0.000, E1  +398.905, E3 -373543.776}
SPL {X  -159.990, Y  +660.353, Z    +0.000, E1  +398.930, E3 -373558.307}
SPL {X  -159.990, Y  +665.703, Z    +0.000, E1  +398.903, E3 -373572.414}
SPL {X  -159.990, Y  +669.966, Z    +0.000, E1  +398.902, E3 -373583.621}
SPL {X  -159.954, Y  +674.895, Z    +0.000, E1  +398.910, E3 -373596.601}
SPL {X  -159.761, Y  +680.061, Z    +0.000, E1  +398.873, E3 -373610.380}
SPL {X  -159.327, Y  +686.045, Z    +0.000, E1  +398.835, E3 -373626.502}
SPL {X  -158.832, Y  +690.714, Z    +0.000, E1  +398.685, E3 -373639.428}
SPL {X  -158.318, Y  +694.567, Z    +0.000, E1  +398.614, E3 -373650.075}
SPL {X  -157.472, Y  +699.775, Z    +0.000, E1  +398.483, E3 -373664.635}
SPL {X  -156.506, Y  +704.705, Z    +0.000, E1  +398.294, E3 -373678.635}
SPL {X  -155.357, Y  +709.721, Z    +0.000, E1  +398.108, E3 -373692.990}
SPL {X  -154.286, Y  +713.838, Z    +0.000, E1  +397.877, E3 -373704.973}
SPL {X  -153.345, Y  +717.131, Z    +0.000, E1  +397.713, E3 -373714.587}
SPL {X  -151.080, Y  +724.146, Z    +0.000, E1  +393.201, E3 -373773.041}
ENDSPLINE

SPLINE
SPL {X  -157.921, Y  +697.149, Z    +0.000, E1  +377.701, E3 -373824.602}
SPL {X  -159.579, Y  +682.959, Z    +0.000, E1  +369.793, E3 -373832.550}
SPL {X  -159.938, Y  +675.561, Z    +0.000, E1  +365.399, E3 -373834.972}
SPL {X  -159.990, Y  +669.910, Z    +0.000, E1  +361.710, E3 -373836.263}
SPL {X  -159.990, Y  +665.465, Z    +0.000, E1  +358.378, E3 -373837.181}
SPL {X  -159.990, Y  +661.791, Z    +0.000, E1  +355.213, E3 -373838.018}
SPL {X  -159.990, Y  +656.991, Z    +0.000, E1  +350.742, E3 -373839.438}
SPL {X  -159.990, Y  +648.067, Z    +0.000, E1  +342.328, E3 -373843.167}
SPL {X  -159.990, Y  +620.451, Z    +0.000, E1  +325.419, E3 -373867.014}
SPL {X  -159.990, Y  +591.256, Z    +0.000, E1  +319.966, E3 -373913.508}
SPL {X  -159.990, Y  +586.740, Z    +0.000, E1  +319.956, E3 -373924.898}
SPL {X  -159.990, Y  +581.814, Z    +0.000, E1  +319.956, E3 -373937.338}
SPL {X  -159.990, Y  +577.274, Z    +0.000, E1  +319.964, E3 -373948.815}
SPL {X  -159.990, Y  +572.933, Z    +0.000, E1  +319.959, E3 -373959.756}
SPL {X  -159.990, Y  +568.504, Z    +0.000, E1  +319.956, E3 -373970.919}
SPL {X  -159.990, Y  +563.189, Z    +0.000, E1  +319.932, E3 -373984.292}
SPL {X  -159.990, Y  +557.707, Z    +0.000, E1  +319.949, E3 -373998.148}
SPL {X  -159.990, Y  +553.571, Z    +0.000, E1  +319.954, E3 -374008.566}
SPL {X  -159.990, Y  +549.413, Z    +0.000, E1  +319.938, E3 -374019.032}
SPL {X  -159.990, Y  +543.439, Z    +0.000, E1  +319.921, E3 -374034.120}
SPL {X  -159.990, Y  +537.213, Z    +0.000, E1  +319.937, E3 -374049.863}
SPL {X  -159.990, Y  +530.667, Z    +0.000, E1  +319.910, E3 -374066.321}
SPL {X  -159.990, Y  +523.984, Z    +0.000, E1  +319.922, E3 -374083.187}
SPL {X  -159.990, Y  +502.378, Z    +0.000, E1  +313.079, E3 -374091.298}
SPL {X  -159.990, Y  +493.568, Z    +0.000, E1  +312.053, E3 -374102.466}
SPL {X  -159.990, Y  +488.437, Z    +0.000, E1  +313.241, E3 -374119.681}
SPL {X  -159.990, Y  +483.955, Z    +0.000, E1  +314.316, E3 -374134.931}
SPL {X  -159.990, Y  +479.762, Z    +0.000, E1  +315.381, E3 -374150.322}
SPL {X  -159.990, Y  +474.562, Z    +0.000, E1  +316.600, E3 -374168.992}
SPL {X  -159.990, Y  +470.788, Z    +0.000, E1  +317.853, E3 -374184.875}
SPL {X  -159.990, Y  +467.944, Z    +0.000, E1  +318.635, E3 -374196.196}
SPL {X  -159.990, Y  +465.057, Z    +0.000, E1  +319.375, E3 -374207.761}
SPL {X  -159.990, Y  +461.409, Z    +0.000, E1  +319.848, E3 -374219.661}
SPL {X  -159.990, Y  +456.934, Z    +0.000, E1  +319.854, E3 -374230.936}
SPL {X  -159.990, Y  +452.940, Z    +0.000, E1  +319.854, E3 -374240.981}
SPL {X  -159.990, Y  +448.856, Z    +0.000, E1  +319.859, E3 -374251.264}
SPL {X  -159.990, Y  +443.741, Z    +0.000, E1  +319.827, E3 -374264.082}
SPL {X  -159.990, Y  +436.703, Z    +0.000, E1  +319.809, E3 -374281.764}
SPL {X  -159.990, Y  +430.690, Z    +0.000, E1  +319.854, E3 -374296.957}
SPL {X  -159.990, Y  +426.145, Z    +0.000, E1  +319.853, E3 -374308.397}
SPL {X  -159.990, Y  +421.880, Z    +0.000, E1  +319.860, E3 -374319.130}
SPL {X  -159.990, Y  +416.246, Z    +0.000, E1  +319.819, E3 -374333.258}
SPL {X  -159.990, Y  +409.936, Z    +0.000, E1  +319.849, E3 -374349.195}
SPL {X  -159.990, Y  +404.988, Z    +0.000, E1  +319.861, E3 -374361.661}
SPL {X  -159.990, Y  +400.535, Z    +0.000, E1  +319.859, E3 -374372.859}
SPL {X  -159.990, Y  +396.024, Z    +0.000, E1  +319.860, E3 -374384.215}
SPL {X  -159.990, Y  +391.614, Z    +0.000, E1  +319.860, E3 -374395.309}
SPL {X  -159.990, Y  +387.212, Z    +0.000, E1  +319.859, E3 -374406.381}
SPL {X  -159.990, Y  +382.743, Z    +0.000, E1  +319.857, E3 -374417.622}
SPL {X  -159.925, Y  +377.946, Z    +0.000, E1  +319.864, E3 -374429.759}
SPL {X  -159.703, Y  +372.915, Z    +0.000, E1  +319.904, E3 -374442.659}
SPL {X  -159.358, Y  +368.290, Z    +0.000, E1  +319.961, E3 -374454.622}
SPL {X  -158.955, Y  +364.333, Z    +0.000, E1  +320.046, E3 -374465.024}
SPL {X  -158.482, Y  +360.589, Z    +0.000, E1  +320.125, E3 -374474.950}
SPL {X  -157.729, Y  +355.695, Z    +0.000, E1  +320.237, E3 -374488.023}
SPL {X  -156.893, Y  +351.173, Z    +0.000, E1  +320.410, E3 -374500.306}
SPL {X  -156.148, Y  +347.650, Z    +0.000, E1  +320.549, E3 -374509.952}
SPL {X  -155.268, Y  +343.918, Z    +0.000, E1  +320.696, E3 -374520.233}
SPL {X  -154.153, Y  +339.677, Z    +0.000, E1  +320.896, E3 -374532.040}
SPL {X  -152.885, Y  +335.352, Z    +0.000, E1  +321.114, E3 -374544.194}
SPL {X  -151.010, Y  +329.654, Z    +0.000, E1  +326.674, E3 -374604.410}
ENDSPLINE

SPLINE
SPL {X  -157.513, Y  +354.453, Z    +0.000, E1  +340.941, E3 -374650.444}
SPL {X  -159.638, Y  +371.886, Z    +0.000, E1  +350.545, E3 -374661.107}
SPL {X  -159.990, Y  +382.357, Z    +0.000, E1  +356.972, E3 -374664.522}
SPL {X  -159.990, Y  +388.001, Z    +0.000, E1  +361.086, E3 -374665.860}
SPL {X  -159.990, Y  +392.647, Z    +0.000, E1  +364.974, E3 -374666.998}
SPL {X  -159.990, Y  +399.434, Z    +0.000, E1  +371.306, E3 -374669.179}
SPL {X  -159.990, Y  +409.375, Z    +0.000, E1  +380.357, E3 -374674.211}
SPL {X  -159.990, Y  +434.822, Z    +0.000, E1  +394.625, E3 -374697.781}
SPL {X  -159.990, Y  +460.330, Z    +0.000, E1  +398.908, E3 -374742.057}
SPL {X  -159.990, Y  +464.953, Z    +0.000, E1  +398.907, E3 -374754.215}
SPL {X  -159.990, Y  +469.353, Z    +0.000, E1  +398.902, E3 -374765.796}
SPL {X  -159.990, Y  +475.034, Z    +0.000, E1  +398.936, E3 -374780.711}
SPL {X  -159.990, Y  +481.308, Z    +0.000, E1  +398.917, E3 -374797.221}
SPL {X  -159.990, Y  +485.396, Z    +0.000, E1  +398.893, E3 -374807.981}
SPL {X  -159.990, Y  +488.362, Z    +0.000, E1  +398.896, E3 -374815.764}
SPL {X  -159.990, Y  +492.629, Z    +0.000, E1  +398.922, E3 -374826.936}
SPL {X  -159.990, Y  +497.431, Z    +0.000, E1  +398.905, E3 -374839.602}
SPL {X  -159.990, Y  +502.093, Z    +0.000, E1  +398.909, E3 -374851.876}
SPL {X  -159.990, Y  +507.821, Z    +0.000, E1  +398.930, E3 -374866.897}
SPL {X  -159.990, Y  +513.533, Z    +0.000, E1  +398.910, E3 -374881.956}
SPL {X  -159.990, Y  +518.435, Z    +0.000, E1  +398.905, E3 -374894.851}
SPL {X  -159.990, Y  +523.478, Z    +0.000, E1  +398.918, E3 -374908.080}
SPL {X  -159.990, Y  +528.627, Z    +0.000, E1  +398.910, E3 -374921.633}
SPL {X  -159.990, Y  +533.053, Z    +0.000, E1  +398.899, E3 -374933.291}
SPL {X  -159.990, Y  +537.174, Z    +0.000, E1  +398.910, E3 -374944.105}
SPL {X  -159.990, Y  +541.259, Z    +0.000, E1  +398.888, E3 -374954.905}
SPL {X  -159.990, Y  +545.676, Z    +0.000, E1  +398.913, E3 -374966.476}
SPL {X  -159.990, Y  +550.777, Z    +0.000, E1  +398.906, E3 -374979.895}
SPL {X  -159.990, Y  +554.638, Z    +0.000, E1  +398.890, E3 -374990.066}
SPL {X  -159.990, Y  +557.678, Z    +0.000, E1  +398.893, E3 -374998.041}
SPL {X  -159.990, Y  +561.696, Z    +0.000, E1  +398.912, E3 -375008.567}
SPL {X  -159.990, Y  +566.650, Z    +0.000, E1  +398.917, E3 -375021.581}
SPL {X  -159.990, Y  +571.814, Z    +0.000, E1  +398.914, E3 -375035.183}
SPL {X  -159.990, Y  +577.636, Z    +0.000, E1  +398.929, E3 -375050.481}
SPL {X  -159.990, Y  +583.167, Z    +0.000, E1  +398.906, E3 -375065.056}
SPL {X  -159.990, Y  +587.761, Z    +0.000, E1  +398.902, E3 -375077.141}
SPL {X  -159.990, Y  +592.962, Z    +0.000, E1  +398.925, E3 -375090.785}
SPL {X  -159.990, Y  +597.767, Z    +0.000, E1  +398.897, E3 -375103.460}
SPL {X  -159.990, Y  +602.727, Z    +0.000, E1  +398.920, E3 -375116.471}
SPL {X  -159.990, Y  +608.112, Z    +0.000, E1  +398.911, E3 -375130.646}
SPL {X  -159.990, Y  +614.125, Z    +0.000, E1  +398.936, E3 -375146.421}
SPL {X  -159.990, Y  +619.061, Z    +0.000, E1  +398.894, E3 -375159.453}
SPL {X  -159.990, Y  +623.264, Z    +0.000, E1  +398.906, E3 -375170.502}
SPL {X  -159.990, Y  +628.669, Z    +0.000, E1  +398.928, E3 -375184.670}
SPL {X  -159.990, Y  +634.089, Z    +0.000, E1  +398.907, E3 -375198.945}
SPL {X  -159.990, Y  +638.639, Z    +0.000, E1  +398.904, E3 -375210.931}
SPL {X  -159.990, Y  +643.555, Z    +0.000, E1  +398.910, E3 -375223.851}
SPL {X  -159.990, Y  +649.380, Z    +0.000, E1  +398.930, E3 -375239.129}
SPL {X  -159.990, Y  +654.813, Z    +0.000, E1  +398.905, E3 -375253.453}
SPL {X  -159.990, Y  +660.353, Z    +0.000, E1  +398.930, E3 -375267.984}
SPL {X  -159.990, Y  +665.703, Z    +0.000, E1  +398.903, E3 -375282.092}
SPL {X  -159.990, Y  +671.472, Z    +0.000, E1  +398.942, E3 -375297.196}
SPL {X  -159.920, Y  +676.216, Z    +0.000, E1  +398.875, E3 -375309.832}
SPL {X  -159.761, Y  +680.061, Z    +0.000, E1  +398.873, E3 -375320.057}
SPL {X  -159.443, Y  +684.716, Z    +0.000, E1  +398.815, E3 -375332.622}
SPL {X  -158.962, Y  +689.604, Z    +0.000, E1  +398.740, E3 -375345.992}
SPL {X  -158.318, Y  +694.567, Z    +0.000, E1  +398.614, E3 -375359.753}
SPL {X  -157.472, Y  +699.775, Z    +0.000, E1  +398.483, E3 -375374.312}
SPL {X  -156.506, Y  +704.705, Z    +0.000, E1  +398.294, E3 -375388.313}
SPL {X  -155.357, Y  +709.721, Z    +0.000, E1  +398.108, E3 -375402.668}
SPL {X  -154.286, Y  +713.838, Z    +0.000, E1  +397.877, E3 -375414.650}
SPL {X  -153.345, Y  +717.131, Z    +0.000, E1  +397.713, E3 -375424.265}
SPL {X  -151.080, Y  +724.146, Z    +0.000, E1  +393.201, E3 -375482.718}
ENDSPLINE

SPLINE
SPL {X  -157.921, Y  +697.149, Z    +0.000, E1  +377.701, E3 -375534.279}
SPL {X  -159.579, Y  +682.959, Z    +0.000, E1  +369.793, E3 -375542.228}
SPL {X  -159.938, Y  +675.561, Z    +0.000, E1  +365.399, E3 -375544.650}
SPL {X  -159.990, Y  +669.910, Z    +0.000, E1  +361.710, E3 -375545.941}
SPL {X  -159.990, Y  +665.465, Z    +0.000, E1  +358.378, E3 -375546.858}
SPL {X  -159.990, Y  +661.791, Z    +0.000, E1  +355.213, E3 -375547.696}
SPL {X  -159.990, Y  +656.991, Z    +0.000, E1  +350.742, E3 -375549.115}
SPL {X  -159.990, Y  +649.722, Z    +0.000, E1  +343.777, E3 -375552.034}
SPL {X  -159.990, Y  +645.752, Z    +0.000, E1  +340.157, E3 -375553.975}
SPL {X  -159.990, Y  +624.891, Z    +0.000, E1  +327.004, E3 -375571.333}
SPL {X  -159.990, Y  +618.109, Z    +0.000, E1  +324.631, E3 -375579.509}
SPL {X  -159.990, Y  +591.256, Z    +0.000, E1  +319.966, E3 -375623.185}
SPL {X  -159.990, Y  +586.740, Z    +0.000, E1  +319.956, E3 -375634.575}
SPL {X  -159.990, Y  +581.814, Z    +0.000, E1  +319.956, E3 -375647.015}
SPL {X  -159.990, Y  +577.274, Z    +0.000, E1  +319.964, E3 -375658.493}
SPL {X  -159.990, Y  +572.933, Z    +0.000, E1  +319.959, E3 -375669.434}
SPL {X  -159.990, Y  +568.504, Z    +0.000, E1  +319.956, E3 -375680.596}
SPL {X  -159.990, Y  +564.427, Z    +0.000, E1  +319.959, E3 -375690.882}
SPL {X  -159.990, Y  +558.823, Z    +0.000, E1  +319.916, E3 -375704.962}
SPL {X  -159.990, Y  +553.571, Z    +0.000, E1  +319.954, E3 -375718.244}
SPL {X  -159.990, Y  +549.413, Z    +0.000, E1  +319.938, E3 -375728.710}
SPL {X  -159.990, Y  +544.924, Z    +0.000, E1  +319.955, E3 -375740.091}
SPL {X  -159.990, Y  +540.054, Z    +0.000, E1  +319.939, E3 -375752.377}
SPL {X  -159.990, Y  +533.683, Z    +0.000, E1  +319.916, E3 -375768.402}
SPL {X  -159.990, Y  +528.899, Z    +0.000, E1  +319.955, E3 -375780.518}
SPL {X  -159.990, Y  +523.984, Z    +0.000, E1  +319.922, E3 -375792.864}
SPL {X  -159.990, Y  +495.402, Z    +0.000, E1  +312.238, E3 -375809.794}
SPL {X  -159.990, Y  +489.464, Z    +0.000, E1  +313.059, E3 -375826.010}
SPL {X  -159.990, Y  +484.831, Z    +0.000, E1  +314.066, E3 -375841.543}
SPL {X  -159.990, Y  +479.762, Z    +0.000, E1  +315.381, E3 -375859.999}
SPL {X  -159.990, Y  +475.871, Z    +0.000, E1  +316.362, E3 -375874.048}
SPL {X  -159.990, Y  +472.671, Z    +0.000, E1  +317.192, E3 -375886.351}
SPL {X  -159.990, Y  +468.809, Z    +0.000, E1  +318.343, E3 -375902.280}
SPL {X  -159.990, Y  +465.057, Z    +0.000, E1  +319.375, E3 -375917.438}
SPL {X  -159.990, Y  +461.409, Z    +0.000, E1  +319.848, E3 -375929.338}
SPL {X  -159.990, Y  +456.934, Z    +0.000, E1  +319.854, E3 -375940.614}
SPL {X  -159.990, Y  +452.940, Z    +0.000, E1  +319.854, E3 -375950.658}
SPL {X  -159.990, Y  +448.856, Z    +0.000, E1  +319.859, E3 -375960.942}
SPL {X  -159.990, Y  +444.973, Z    +0.000, E1  +319.856, E3 -375970.707}
SPL {X  -159.990, Y  +439.927, Z    +0.000, E1  +319.837, E3 -375983.363}
SPL {X  -159.990, Y  +435.246, Z    +0.000, E1  +319.853, E3 -375995.173}
SPL {X  -159.990, Y  +430.690, Z    +0.000, E1  +319.854, E3 -376006.634}
SPL {X  -159.990, Y  +426.145, Z    +0.000, E1  +319.853, E3 -376018.074}
SPL {X  -159.990, Y  +421.880, Z    +0.000, E1  +319.860, E3 -376028.807}
SPL {X  -159.990, Y  +417.572, Z    +0.000, E1  +319.852, E3 -376039.634}
SPL {X  -159.990, Y  +412.619, Z    +0.000, E1  +319.850, E3 -376052.125}
SPL {X  -159.990, Y  +406.264, Z    +0.000, E1  +319.825, E3 -376068.074}
SPL {X  -159.990, Y  +400.535, Z    +0.000, E1  +319.859, E3 -376082.536}
SPL {X  -159.990, Y  +396.024, Z    +0.000, E1  +319.860, E3 -376093.892}
SPL {X  -159.990, Y  +391.614, Z    +0.000, E1  +319.860, E3 -376104.986}
SPL {X  -159.990, Y  +387.212, Z    +0.000, E1  +319.859, E3 -376116.058}
SPL {X  -159.990, Y  +382.743, Z    +0.000, E1  +319.857, E3 -376127.300}
SPL {X  -159.925, Y  +377.946, Z    +0.000, E1  +319.864, E3 -376139.437}
SPL {X  -159.703, Y  +372.915, Z    +0.000, E1  +319.904, E3 -376152.336}
SPL {X  -159.358, Y  +368.290, Z    +0.000, E1  +319.961, E3 -376164.299}
SPL {X  -158.955, Y  +364.333, Z    +0.000, E1  +320.046, E3 -376174.701}
SPL {X  -158.482, Y  +360.589, Z    +0.000, E1  +320.125, E3 -376184.628}
SPL {X  -157.729, Y  +355.695, Z    +0.000, E1  +320.237, E3 -376197.700}
SPL {X  -156.893, Y  +351.173, Z    +0.000, E1  +320.410, E3 -376209.984}
SPL {X  -156.148, Y  +347.650, Z    +0.000, E1  +320.549, E3 -376219.630}
SPL {X  -155.268, Y  +343.918, Z    +0.000, E1  +320.696, E3 -376229.910}
SPL {X  -153.936, Y  +338.906, Z    +0.000, E1  +320.911, E3 -376243.850}
SPL {X  -152.628, Y  +334.526, Z    +0.000, E1  +321.188, E3 -376256.252}
SPL {X  -151.010, Y  +329.654, Z    +0.000, E1  +326.674, E3 -376314.088}
ENDSPLINE

